LIN {X 0,Y 106.978,Z 615.98,A -85,B 0,C 180,E1 -26170.823,E2 -26170.823} C_VEL
LIN {X 0,Y 105.342,Z 616.584,A -85,B 0,C 180,E1 -26178.454,E2 -26178.454} C_VEL
LIN {X 0,Y 105.049,Z 615.86,A -85,B 0,C 180,E1 -26186.164,E2 -26186.164} C_VEL
LIN {X 0,Y 105.656,Z 613.825,A -85,B 0,C 180,E1 -26193.814,E2 -26193.814} C_VEL
LIN {X 0,Y 107.51,Z 610.427,A -85,B 0,C 180,E1 -26201.31,E2 -26201.31} C_VEL
LIN {X 0,Y 109.983,Z 606.946,A -85,B 0,C 180,E1 -26206.711,E2 -26206.711} C_VEL
LIN {X 0,Y 113.032,Z 602.521,A -85,B 0,C 180,E1 -26211.905,E2 -26211.905} C_VEL
LIN {X 0,Y 116.825,Z 597.145,A -85,B 0,C 180,E1 -26216.82,E2 -26216.82} C_VEL
LIN {X 0,Y 122.258,Z 589.447,A -85,B 0,C 180,E1 -26222.123,E2 -26222.123} C_VEL
LIN {X 0,Y 127.809,Z 581.397,A -85,B 0,C 180,E1 -26226.237,E2 -26226.237} C_VEL
LIN {X 0,Y 133.781,Z 571.709,A -85,B 0,C 180,E1 -26230.056,E2 -26230.056} C_VEL
LIN {X 0,Y 139.018,Z 562.033,A -85,B 0,C 180,E1 -26233.039,E2 -26233.039} C_VEL
LIN {X 0,Y 142.904,Z 554.154,A -85,B 0,C 180,E1 -26234.988,E2 -26234.988} C_VEL
LIN {X 0,Y 148.241,Z 542.028,A -85,B 0,C 180,E1 -26237.294,E2 -26237.294} C_VEL
LIN {X 0,Y 152.497,Z 530.39,A -85,B 0,C 180,E1 -26238.996,E2 -26238.996} C_VEL
LIN {X 0,Y 156.549,Z 516.515,A -85,B 0,C 180,E1 -26240.498,E2 -26240.498} C_VEL
LIN {X 0,Y 159.485,Z 502.683,A -85,B 0,C 180,E1 -26241.588,E2 -26241.588} C_VEL
LIN {X 0,Y 161.455,Z 488.768,A -85,B 0,C 180,E1 -26242.305,E2 -26242.305} C_VEL
LIN {X 0,Y 165.188,Z 446.212,A -85,B 0,C 180,E1 -26243.697,E2 -26243.697} C_VEL
LIN {X 0,Y 164.983,Z 444.977,A -85,B 0,C 180,E1 -26243.9,E2 -26243.9} C_VEL
LIN {X 0,Y 160.619,Z 435.797,A -85,B 0,C 180,E1 -26247.142,E2 -26247.142} C_VEL
LIN {X 0,Y 155.978,Z 427.263,A -85,B 0,C 180,E1 -26251.089,E2 -26251.089} C_VEL
LIN {X 0,Y 152.792,Z 421.962,A -85,B 0,C 180,E1 -26254.257,E2 -26254.257} C_VEL
LIN {X 0,Y 151.006,Z 419.154,A -85,B 0,C 180,E1 -26256.274,E2 -26256.274} C_VEL
LIN {X 0,Y 148.875,Z 415.814,A -85,B 0,C 180,E1 -26259.026,E2 -26259.026} C_VEL
LIN {X 0,Y 146.603,Z 412.142,A -85,B 0,C 180,E1 -26262.627,E2 -26262.627} C_VEL
LIN {X 0,Y 144.109,Z 408.852,A -85,B 0,C 180,E1 -26268.036,E2 -26268.036} C_VEL
LIN {X 0,Y 143.541,Z 407.096,A -85,B 0,C 180,E1 -26270.22,E2 -26270.22} C_VEL
LIN {X 0,Y 142.692,Z 406.337,A -85,B 0,C 180,E1 -26279.999,E2 -26279.999} C_VEL
LIN {X 0,Y 143.838,Z 407.423,A -85,B 0,C 180,E1 -26285.431,E2 -26285.431} C_VEL
LIN {X 0,Y 145.342,Z 410.732,A -85,B 0,C 180,E1 -26289.655,E2 -26289.655} C_VEL
LIN {X 0,Y 146.816,Z 412.43,A -85,B 0,C 180,E1 -26292.379,E2 -26292.379} C_VEL
LIN {X 0,Y 149.795,Z 417.149,A -85,B 0,C 180,E1 -26296.842,E2 -26296.842} C_VEL
LIN {X 0,Y 152.53,Z 421.521,A -85,B 0,C 180,E1 -26300.095,E2 -26300.095} C_VEL
LIN {X 0,Y 156.091,Z 427.345,A -85,B 0,C 180,E1 -26303.64,E2 -26303.64} C_VEL
LIN {X 0,Y 159.027,Z 432.919,A -85,B 0,C 180,E1 -26306.227,E2 -26306.227} C_VEL
LIN {X 0,Y 161.926,Z 440.414,A -85,B 0,C 180,E1 -26308.674,E2 -26308.674} C_VEL
LIN {X 0,Y 164.965,Z 449.328,A -85,B 0,C 180,E1 -26311.066,E2 -26311.066} C_VEL
LIN {X 0,Y 160.741,Z 497.527,A -85,B 0,C 180,E1 -26312.71,E2 -26312.71} C_VEL
LIN {X 0,Y 158.258,Z 511.944,A -85,B 0,C 180,E1 -26313.483,E2 -26313.483} C_VEL
LIN {X 0,Y 154.769,Z 525.923,A -85,B 0,C 180,E1 -26314.609,E2 -26314.609} C_VEL
LIN {X 0,Y 150.269,Z 539.82,A -85,B 0,C 180,E1 -26316.218,E2 -26316.218} C_VEL
LIN {X 0,Y 145.255,Z 552.264,A -85,B 0,C 180,E1 -26318.164,E2 -26318.164} C_VEL
LIN {X 0,Y 139.927,Z 563.656,A -85,B 0,C 180,E1 -26320.564,E2 -26320.564} C_VEL
LIN {X 0,Y 134.889,Z 573.146,A -85,B 0,C 180,E1 -26323.161,E2 -26323.161} C_VEL
LIN {X 0,Y 128.511,Z 583.722,A -85,B 0,C 180,E1 -26326.874,E2 -26326.874} C_VEL
LIN {X 0,Y 122.736,Z 592.445,A -85,B 0,C 180,E1 -26330.959,E2 -26330.959} C_VEL
LIN {X 0,Y 116.945,Z 600.809,A -85,B 0,C 180,E1 -26336.228,E2 -26336.228} C_VEL
LIN {X 0,Y 112.321,Z 607.529,A -85,B 0,C 180,E1 -26342.012,E2 -26342.012} C_VEL
LIN {X 0,Y 108.35,Z 613.483,A -85,B 0,C 180,E1 -26349.099,E2 -26349.099} C_VEL
LIN {X 0,Y 106.4,Z 616.926,A -85,B 0,C 180,E1 -26354.68,E2 -26354.68} C_VEL
LIN {X 0,Y 105.166,Z 620.167,A -85,B 0,C 180,E1 -26362.319,E2 -26362.319} C_VEL
LIN {X 0,Y 105.166,Z 622,A -85,B 0,C 180,E1 -26370,E2 -26370} C_VEL
LIN {X 0,Y 105.173,Z 622.449,A -85,B 0,C 180,E1 -26377.681,E2 -26377.681} C_VEL
LIN {X 0,Y 106.49,Z 621.572,A -85,B 0,C 180,E1 -26385.307,E2 -26385.307} C_VEL
LIN {X 0,Y 109.442,Z 619.368,A -85,B 0,C 180,E1 -26392.663,E2 -26392.663} C_VEL
LIN {X 0,Y 113.967,Z 615.782,A -85,B 0,C 180,E1 -26399.561,E2 -26399.561} C_VEL
LIN {X 0,Y 115.217,Z 614.69,A -85,B 0,C 180,E1 -26401.159,E2 -26401.159} C_VEL
LIN {X 0,Y 116.887,Z 612.823,A -85,B 0,C 180,E1 -26403.808,E2 -26403.808} C_VEL
LIN {X 0,Y 118.627,Z 609.391,A -85,B 0,C 180,E1 -26408.262,E2 -26408.262} C_VEL
LIN {X 0,Y 120.996,Z 605.387,A -85,B 0,C 180,E1 -26412.441,E2 -26412.441} C_VEL
LIN {X 0,Y 123.544,Z 602.626,A -85,B 0,C 180,E1 -26414.574,E2 -26414.574} C_VEL
LIN {X 0,Y 131.067,Z 595.341,A -85,B 0,C 180,E1 -26418.652,E2 -26418.652} C_VEL
LIN {X 0,Y 138.379,Z 587.385,A -85,B 0,C 180,E1 -26421.926,E2 -26421.926} C_VEL
LIN {X 0,Y 146.072,Z 577.81,A -85,B 0,C 180,E1 -26424.879,E2 -26424.879} C_VEL
LIN {X 0,Y 153.417,Z 567.213,A -85,B 0,C 180,E1 -26427.327,E2 -26427.327} C_VEL
LIN {X 0,Y 160.399,Z 555.509,A -85,B 0,C 180,E1 -26429.305,E2 -26429.305} C_VEL
LIN {X 0,Y 166.846,Z 542.503,A -85,B 0,C 180,E1 -26430.933,E2 -26430.933} C_VEL
LIN {X 0,Y 172,Z 529.708,A -85,B 0,C 180,E1 -26432.082,E2 -26432.082} C_VEL
LIN {X 0,Y 176.163,Z 516.241,A -85,B 0,C 180,E1 -26432.995,E2 -26432.995} C_VEL
LIN {X 0,Y 179.308,Z 502.034,A -85,B 0,C 180,E1 -26433.65,E2 -26433.65} C_VEL
LIN {X 0,Y 181.338,Z 486.524,A -85,B 0,C 180,E1 -26434.126,E2 -26434.126} C_VEL
LIN {X 0,Y 182.905,Z 469.902,A -85,B 0,C 180,E1 -26434.606,E2 -26434.606} C_VEL
LIN {X 0,Y 180.192,Z 461.706,A -85,B 0,C 180,E1 -26437.618,E2 -26437.618} C_VEL
LIN {X 0,Y 177.811,Z 455.265,A -85,B 0,C 180,E1 -26440.67,E2 -26440.67} C_VEL
LIN {X 0,Y 175.542,Z 451.014,A -85,B 0,C 180,E1 -26443.967,E2 -26443.967} C_VEL
LIN {X 0,Y 174.032,Z 448.052,A -85,B 0,C 180,E1 -26446.779,E2 -26446.779} C_VEL
LIN {X 0,Y 172.41,Z 444.514,A -85,B 0,C 180,E1 -26451.208,E2 -26451.208} C_VEL
LIN {X 0,Y 171.43,Z 443.369,A -85,B 0,C 180,E1 -26457.651,E2 -26457.651} C_VEL
LIN {X 0,Y 171.628,Z 443.532,A -85,B 0,C 180,E1 -26460.587,E2 -26460.587} C_VEL
LIN {X 0,Y 172.488,Z 444.731,A -85,B 0,C 180,E1 -26464.529,E2 -26464.529} C_VEL
LIN {X 0,Y 174.188,Z 448.243,A -85,B 0,C 180,E1 -26468.959,E2 -26468.959} C_VEL
LIN {X 0,Y 176.521,Z 452.894,A -85,B 0,C 180,E1 -26472.997,E2 -26472.997} C_VEL
LIN {X 0,Y 179.277,Z 458.182,A -85,B 0,C 180,E1 -26476.586,E2 -26476.586} C_VEL
LIN {X 0,Y 182.826,Z 465.868,A -85,B 0,C 180,E1 -26480.376,E2 -26480.376} C_VEL
LIN {X 0,Y 183.217,Z 466.787,A -85,B 0,C 180,E1 -26480.756,E2 -26480.756} C_VEL
LIN {X 0,Y 180.381,Z 493.857,A -85,B 0,C 180,E1 -26481.549,E2 -26481.549} C_VEL
LIN {X 0,Y 177.612,Z 508.239,A -85,B 0,C 180,E1 -26482.207,E2 -26482.207} C_VEL
LIN {X 0,Y 173.834,Z 521.809,A -85,B 0,C 180,E1 -26483.106,E2 -26483.106} C_VEL
LIN {X 0,Y 168.725,Z 535.471,A -85,B 0,C 180,E1 -26484.295,E2 -26484.295} C_VEL
LIN {X 0,Y 163.676,Z 546.452,A -85,B 0,C 180,E1 -26485.615,E2 -26485.615} C_VEL
LIN {X 0,Y 157.42,Z 557.978,A -85,B 0,C 180,E1 -26487.461,E2 -26487.461} C_VEL
LIN {X 0,Y 151.225,Z 567.55,A -85,B 0,C 180,E1 -26489.379,E2 -26489.379} C_VEL
LIN {X 0,Y 144.635,Z 576.544,A -85,B 0,C 180,E1 -26491.75,E2 -26491.75} C_VEL
LIN {X 0,Y 137.144,Z 585.567,A -85,B 0,C 180,E1 -26494.922,E2 -26494.922} C_VEL
LIN {X 0,Y 128.837,Z 594.174,A -85,B 0,C 180,E1 -26498.982,E2 -26498.982} C_VEL
LIN {X 0,Y 121.282,Z 601.093,A -85,B 0,C 180,E1 -26503.588,E2 -26503.588} C_VEL
LIN {X 0,Y 115.515,Z 605.855,A -85,B 0,C 180,E1 -26507.991,E2 -26507.991} C_VEL
LIN {X 0,Y 108.934,Z 610.764,A -85,B 0,C 180,E1 -26514.504,E2 -26514.504} C_VEL
LIN {X 0,Y 103.848,Z 614.157,A -85,B 0,C 180,E1 -26521.723,E2 -26521.723} C_VEL
LIN {X 0,Y 100.215,Z 616.148,A -85,B 0,C 180,E1 -26529.473,E2 -26529.473} C_VEL
LIN {X 0,Y 98.338,Z 616.788,A -85,B 0,C 180,E1 -26537.619,E2 -26537.619} C_VEL
LIN {X 0,Y 97.939,Z 616.099,A -85,B 0,C 180,E1 -26545.885,E2 -26545.885} C_VEL
LIN {X 0,Y 98.14,Z 615.26,A -85,B 0,C 180,E1 -26550,E2 -26550} C_VEL
LIN {X 0,Y 99.433,Z 612.582,A -85,B 0,C 180,E1 -26558.127,E2 -26558.127} C_VEL
LIN {X 0,Y 102.251,Z 608.494,A -85,B 0,C 180,E1 -26565.958,E2 -26565.958} C_VEL
LIN {X 0,Y 105.321,Z 604.462,A -85,B 0,C 180,E1 -26571.531,E2 -26571.531} C_VEL
LIN {X 0,Y 109.144,Z 599.427,A -85,B 0,C 180,E1 -26576.791,E2 -26576.791} C_VEL
LIN {X 0,Y 114.497,Z 592.249,A -85,B 0,C 180,E1 -26582.486,E2 -26582.486} C_VEL
LIN {X 0,Y 121.199,Z 583.338,A -85,B 0,C 180,E1 -26587.508,E2 -26587.508} C_VEL
LIN {X 0,Y 127.323,Z 574.006,A -85,B 0,C 180,E1 -26591.482,E2 -26591.482} C_VEL
LIN {X 0,Y 133.326,Z 563.687,A -85,B 0,C 180,E1 -26594.833,E2 -26594.833} C_VEL
LIN {X 0,Y 137.993,Z 554.781,A -85,B 0,C 180,E1 -26597.065,E2 -26597.065} C_VEL
LIN {X 0,Y 143.54,Z 542.777,A -85,B 0,C 180,E1 -26599.369,E2 -26599.369} C_VEL
LIN {X 0,Y 147.966,Z 531.241,A -85,B 0,C 180,E1 -26601.057,E2 -26601.057} C_VEL
LIN {X 0,Y 152.165,Z 517.653,A -85,B 0,C 180,E1 -26602.546,E2 -26602.546} C_VEL
LIN {X 0,Y 155.378,Z 503.296,A -85,B 0,C 180,E1 -26603.677,E2 -26603.677} C_VEL
LIN {X 0,Y 157.437,Z 489.422,A -85,B 0,C 180,E1 -26604.398,E2 -26604.398} C_VEL
LIN {X 0,Y 161.101,Z 449.238,A -85,B 0,C 180,E1 -26605.705,E2 -26605.705} C_VEL
LIN {X 0,Y 160.919,Z 447.991,A -85,B 0,C 180,E1 -26605.916,E2 -26605.916} C_VEL
LIN {X 0,Y 156.872,Z 439.376,A -85,B 0,C 180,E1 -26609.251,E2 -26609.251} C_VEL
LIN {X 0,Y 153.029,Z 432.072,A -85,B 0,C 180,E1 -26612.894,E2 -26612.894} C_VEL
LIN {X 0,Y 149.801,Z 426.345,A -85,B 0,C 180,E1 -26616.534,E2 -26616.534} C_VEL
LIN {X 0,Y 147.291,Z 422.35,A -85,B 0,C 180,E1 -26619.918,E2 -26619.918} C_VEL
LIN {X 0,Y 145.022,Z 418.618,A -85,B 0,C 180,E1 -26623.819,E2 -26623.819} C_VEL
LIN {X 0,Y 142.956,Z 415.552,A -85,B 0,C 180,E1 -26628.854,E2 -26628.854} C_VEL
LIN {X 0,Y 142.531,Z 414.075,A -85,B 0,C 180,E1 -26630.707,E2 -26630.707} C_VEL
LIN {X 0,Y 141.824,Z 413.393,A -85,B 0,C 180,E1 -26639.999,E2 -26639.999} C_VEL
LIN {X 0,Y 142.761,Z 414.272,A -85,B 0,C 180,E1 -26644.764,E2 -26644.764} C_VEL
LIN {X 0,Y 144.362,Z 417.845,A -85,B 0,C 180,E1 -26649.5,E2 -26649.5} C_VEL
LIN {X 0,Y 145.476,Z 419.202,A -85,B 0,C 180,E1 -26651.661,E2 -26651.661} C_VEL
LIN {X 0,Y 148.187,Z 423.711,A -85,B 0,C 180,E1 -26656.001,E2 -26656.001} C_VEL
LIN {X 0,Y 150.663,Z 427.94,A -85,B 0,C 180,E1 -26659.157,E2 -26659.157} C_VEL
LIN {X 0,Y 153.786,Z 433.303,A -85,B 0,C 180,E1 -26662.492,E2 -26662.492} C_VEL
LIN {X 0,Y 156.38,Z 438.493,A -85,B 0,C 180,E1 -26664.959,E2 -26664.959} C_VEL
LIN {X 0,Y 159.939,Z 448.587,A -85,B 0,C 180,E1 -26668.192,E2 -26668.192} C_VEL
LIN {X 0,Y 160.916,Z 451.729,A -85,B 0,C 180,E1 -26669.034,E2 -26669.034} C_VEL
LIN {X 0,Y 156.748,Z 497.427,A -85,B 0,C 180,E1 -26670.589,E2 -26670.589} C_VEL
LIN {X 0,Y 154.257,Z 511.481,A -85,B 0,C 180,E1 -26671.322,E2 -26671.322} C_VEL
LIN {X 0,Y 150.816,Z 524.958,A -85,B 0,C 180,E1 -26672.368,E2 -26672.368} C_VEL
LIN {X 0,Y 146.84,Z 537.25,A -85,B 0,C 180,E1 -26673.736,E2 -26673.736} C_VEL
LIN {X 0,Y 141.6,Z 550.147,A -85,B 0,C 180,E1 -26675.635,E2 -26675.635} C_VEL
LIN {X 0,Y 135.961,Z 561.87,A -85,B 0,C 180,E1 -26677.974,E2 -26677.974} C_VEL
LIN {X 0,Y 130.121,Z 572.617,A -85,B 0,C 180,E1 -26680.873,E2 -26680.873} C_VEL
LIN {X 0,Y 123.378,Z 583.245,A -85,B 0,C 180,E1 -26684.599,E2 -26684.599} C_VEL
LIN {X 0,Y 117.257,Z 592.014,A -85,B 0,C 180,E1 -26688.753,E2 -26688.753} C_VEL
LIN {X 0,Y 111.066,Z 600.428,A -85,B 0,C 180,E1 -26694.175,E2 -26694.175} C_VEL
LIN {X 0,Y 106.029,Z 607.187,A -85,B 0,C 180,E1 -26700.19,E2 -26700.19} C_VEL
LIN {X 0,Y 101.712,Z 613.176,A -85,B 0,C 180,E1 -26707.664,E2 -26707.664} C_VEL
LIN {X 0,Y 99.515,Z 616.637,A -85,B 0,C 180,E1 -26713.591,E2 -26713.591} C_VEL
LIN {X 0,Y 98.102,Z 619.917,A -85,B 0,C 180,E1 -26721.762,E2 -26721.762} C_VEL
LIN {X 0,Y 98.072,Z 621.779,A -85,B 0,C 180,E1 -26730,E2 -26730} C_VEL
LIN {X 0,Y 98.113,Z 622.254,A -85,B 0,C 180,E1 -26738.237,E2 -26738.237} C_VEL
LIN {X 0,Y 99.624,Z 621.403,A -85,B 0,C 180,E1 -26746.391,E2 -26746.391} C_VEL
LIN {X 0,Y 102.883,Z 619.226,A -85,B 0,C 180,E1 -26754.197,E2 -26754.197} C_VEL
LIN {X 0,Y 107.79,Z 615.668,A -85,B 0,C 180,E1 -26761.441,E2 -26761.441} C_VEL
LIN {X 0,Y 114.247,Z 610.629,A -85,B 0,C 180,E1 -26767.964,E2 -26767.964} C_VEL
LIN {X 0,Y 122.109,Z 603.966,A -85,B 0,C 180,E1 -26773.683,E2 -26773.683} C_VEL
LIN {X 0,Y 123.544,Z 602.626,A -85,B 0,C 180,E1 -26774.574,E2 -26774.574} C_VEL
LIN {X 0,Y 126.194,Z 599.722,A -85,B 0,C 180,E1 -26776.597,E2 -26776.597} C_VEL
LIN {X 0,Y 129.378,Z 594.686,A -85,B 0,C 180,E1 -26780.169,E2 -26780.169} C_VEL
LIN {X 0,Y 132.837,Z 589.224,A -85,B 0,C 180,E1 -26783.445,E2 -26783.445} C_VEL
LIN {X 0,Y 135.79,Z 585.532,A -85,B 0,C 180,E1 -26784.964,E2 -26784.964} C_VEL
LIN {X 0,Y 143.447,Z 576.129,A -85,B 0,C 180,E1 -26787.688,E2 -26787.688} C_VEL
LIN {X 0,Y 151.134,Z 565.237,A -85,B 0,C 180,E1 -26790.009,E2 -26790.009} C_VEL
LIN {X 0,Y 158.342,Z 553.168,A -85,B 0,C 180,E1 -26791.904,E2 -26791.904} C_VEL
LIN {X 0,Y 164.288,Z 541.252,A -85,B 0,C 180,E1 -26793.254,E2 -26793.254} C_VEL
LIN {X 0,Y 169.568,Z 528.127,A -85,B 0,C 180,E1 -26794.352,E2 -26794.352} C_VEL
LIN {X 0,Y 173.757,Z 514.407,A -85,B 0,C 180,E1 -26795.203,E2 -26795.203} C_VEL
LIN {X 0,Y 176.793,Z 500.293,A -85,B 0,C 180,E1 -26795.815,E2 -26795.815} C_VEL
LIN {X 0,Y 179.048,Z 482.171,A -85,B 0,C 180,E1 -26796.322,E2 -26796.322} C_VEL
LIN {X 0,Y 179.924,Z 473.211,A -85,B 0,C 180,E1 -26796.571,E2 -26796.571} C_VEL
LIN {X 0,Y 177.487,Z 465.387,A -85,B 0,C 180,E1 -26799.672,E2 -26799.672} C_VEL
LIN {X 0,Y 175.976,Z 461.216,A -85,B 0,C 180,E1 -26801.839,E2 -26801.839} C_VEL
LIN {X 0,Y 174.1,Z 457.474,A -85,B 0,C 180,E1 -26804.832,E2 -26804.832} C_VEL
LIN {X 0,Y 172.836,Z 454.794,A -85,B 0,C 180,E1 -26807.399,E2 -26807.399} C_VEL
LIN {X 0,Y 171.379,Z 451.415,A -85,B 0,C 180,E1 -26811.748,E2 -26811.748} C_VEL
LIN {X 0,Y 170.563,Z 450.423,A -85,B 0,C 180,E1 -26817.639,E2 -26817.639} C_VEL
LIN {X 0,Y 170.757,Z 450.614,A -85,B 0,C 180,E1 -26820.59,E2 -26820.59} C_VEL
LIN {X 0,Y 171.482,Z 451.693,A -85,B 0,C 180,E1 -26824.114,E2 -26824.114} C_VEL
LIN {X 0,Y 173.28,Z 455.722,A -85,B 0,C 180,E1 -26829.006,E2 -26829.006} C_VEL
LIN {X 0,Y 175.2,Z 459.749,A -85,B 0,C 180,E1 -26832.452,E2 -26832.452} C_VEL
LIN {X 0,Y 177.515,Z 464.469,A -85,B 0,C 180,E1 -26835.676,E2 -26835.676} C_VEL
LIN {X 0,Y 180.167,Z 470.555,A -85,B 0,C 180,E1 -26838.778,E2 -26838.778} C_VEL
LIN {X 0,Y 177.56,Z 494.301,A -85,B 0,C 180,E1 -26839.467,E2 -26839.467} C_VEL
LIN {X 0,Y 174.687,Z 508.753,A -85,B 0,C 180,E1 -26840.114,E2 -26840.114} C_VEL
LIN {X 0,Y 170.779,Z 522.33,A -85,B 0,C 180,E1 -26840.987,E2 -26840.987} C_VEL
LIN {X 0,Y 165.81,Z 535.301,A -85,B 0,C 180,E1 -26842.079,E2 -26842.079} C_VEL
LIN {X 0,Y 159.976,Z 547.572,A -85,B 0,C 180,E1 -26843.497,E2 -26843.497} C_VEL
LIN {X 0,Y 153.533,Z 558.935,A -85,B 0,C 180,E1 -26845.302,E2 -26845.302} C_VEL
LIN {X 0,Y 146.433,Z 569.358,A -85,B 0,C 180,E1 -26847.388,E2 -26847.388} C_VEL
LIN {X 0,Y 138.319,Z 579.704,A -85,B 0,C 180,E1 -26850.256,E2 -26850.256} C_VEL
LIN {X 0,Y 130.633,Z 588.224,A -85,B 0,C 180,E1 -26853.498,E2 -26853.498} C_VEL
LIN {X 0,Y 122.068,Z 596.332,A -85,B 0,C 180,E1 -26857.659,E2 -26857.659} C_VEL
LIN {X 0,Y 113.892,Z 603.166,A -85,B 0,C 180,E1 -26862.75,E2 -26862.75} C_VEL
LIN {X 0,Y 106.518,Z 608.597,A -85,B 0,C 180,E1 -26868.715,E2 -26868.715} C_VEL
LIN {X 0,Y 100.144,Z 612.764,A -85,B 0,C 180,E1 -26875.845,E2 -26875.845} C_VEL
LIN {X 0,Y 95.319,Z 615.476,A -85,B 0,C 180,E1 -26883.743,E2 -26883.743} C_VEL
LIN {X 0,Y 92.168,Z 616.819,A -85,B 0,C 180,E1 -26892.241,E2 -26892.241} C_VEL
LIN {X 0,Y 90.928,Z 616.826,A -85,B 0,C 180,E1 -26901.107,E2 -26901.107} C_VEL
LIN {X 0,Y 90.828,Z 616.334,A -85,B 0,C 180,E1 -26905.562,E2 -26905.562} C_VEL
LIN {X 0,Y 91.044,Z 615.512,A -85,B 0,C 180,E1 -26910,E2 -26910} C_VEL
LIN {X 0,Y 92.441,Z 612.864,A -85,B 0,C 180,E1 -26918.746,E2 -26918.746} C_VEL
LIN {X 0,Y 95.457,Z 608.807,A -85,B 0,C 180,E1 -26927.128,E2 -26927.128} C_VEL
LIN {X 0,Y 98.764,Z 604.799,A -85,B 0,C 180,E1 -26933.04,E2 -26933.04} C_VEL
LIN {X 0,Y 102.861,Z 599.792,A -85,B 0,C 180,E1 -26938.573,E2 -26938.573} C_VEL
LIN {X 0,Y 108.598,Z 592.652,A -85,B 0,C 180,E1 -26944.49,E2 -26944.49} C_VEL
LIN {X 0,Y 115.681,Z 583.797,A -85,B 0,C 180,E1 -26949.636,E2 -26949.636} C_VEL
LIN {X 0,Y 122.122,Z 574.527,A -85,B 0,C 180,E1 -26953.677,E2 -26953.677} C_VEL
LIN {X 0,Y 128.41,Z 564.276,A -85,B 0,C 180,E1 -26957.057,E2 -26957.057} C_VEL
LIN {X 0,Y 133.278,Z 555.407,A -85,B 0,C 180,E1 -26959.29,E2 -26959.29} C_VEL
LIN {X 0,Y 139.05,Z 543.498,A -85,B 0,C 180,E1 -26961.575,E2 -26961.575} C_VEL
LIN {X 0,Y 143.635,Z 532.081,A -85,B 0,C 180,E1 -26963.247,E2 -26963.247} C_VEL
LIN {X 0,Y 147.98,Z 518.717,A -85,B 0,C 180,E1 -26964.715,E2 -26964.715} C_VEL
LIN {X 0,Y 151.315,Z 504.817,A -85,B 0,C 180,E1 -26965.825,E2 -26965.825} C_VEL
LIN {X 0,Y 153.645,Z 490.117,A -85,B 0,C 180,E1 -26966.59,E2 -26966.59} C_VEL
LIN {X 0,Y 157.258,Z 451.619,A -85,B 0,C 180,E1 -26967.851,E2 -26967.851} C_VEL
LIN {X 0,Y 153.572,Z 443.488,A -85,B 0,C 180,E1 -26971.231,E2 -26971.231} C_VEL
LIN {X 0,Y 149.74,Z 435.854,A -85,B 0,C 180,E1 -26975.362,E2 -26975.362} C_VEL
LIN {X 0,Y 147.457,Z 431.908,A -85,B 0,C 180,E1 -26978.258,E2 -26978.258} C_VEL
LIN {X 0,Y 145.816,Z 428.996,A -85,B 0,C 180,E1 -26980.714,E2 -26980.714} C_VEL
LIN {X 0,Y 143.639,Z 425.279,A -85,B 0,C 180,E1 -26984.752,E2 -26984.752} C_VEL
LIN {X 0,Y 141.841,Z 422.276,A -85,B 0,C 180,E1 -26989.652,E2 -26989.652} C_VEL
LIN {X 0,Y 141.478,Z 421.011,A -85,B 0,C 180,E1 -26991.429,E2 -26991.429} C_VEL
LIN {X 0,Y 140.955,Z 420.453,A -85,B 0,C 180,E1 -26999.999,E2 -26999.999} C_VEL
LIN {X 0,Y 141.765,Z 421.374,A -85,B 0,C 180,E1 -27004.397,E2 -27004.397} C_VEL
LIN {X 0,Y 143.385,Z 424.945,A -85,B 0,C 180,E1 -27009.343,E2 -27009.343} C_VEL
LIN {X 0,Y 144.137,Z 425.963,A -85,B 0,C 180,E1 -27010.89,E2 -27010.89} C_VEL
LIN {X 0,Y 146.71,Z 430.515,A -85,B 0,C 180,E1 -27015.298,E2 -27015.298} C_VEL
LIN {X 0,Y 148.93,Z 434.483,A -85,B 0,C 180,E1 -27018.306,E2 -27018.306} C_VEL
LIN {X 0,Y 152.01,Z 440.251,A -85,B 0,C 180,E1 -27021.813,E2 -27021.813} C_VEL
LIN {X 0,Y 153.809,Z 444.149,A -85,B 0,C 180,E1 -27023.655,E2 -27023.655} C_VEL
LIN {X 0,Y 156.887,Z 453.647,A -85,B 0,C 180,E1 -27026.731,E2 -27026.731} C_VEL
LIN {X 0,Y 157.108,Z 454.381,A -85,B 0,C 180,E1 -27026.942,E2 -27026.942} C_VEL
LIN {X 0,Y 152.938,Z 497.627,A -85,B 0,C 180,E1 -27028.374,E2 -27028.374} C_VEL
LIN {X 0,Y 150.319,Z 511.787,A -85,B 0,C 180,E1 -27029.106,E2 -27029.106} C_VEL
LIN {X 0,Y 146.772,Z 525.133,A -85,B 0,C 180,E1 -27030.128,E2 -27030.128} C_VEL
LIN {X 0,Y 142.317,Z 538.232,A -85,B 0,C 180,E1 -27031.586,E2 -27031.586} C_VEL
LIN {X 0,Y 136.898,Z 550.901,A -85,B 0,C 180,E1 -27033.463,E2 -27033.463} C_VEL
LIN {X 0,Y 131.045,Z 562.456,A -85,B 0,C 180,E1 -27035.79,E2 -27035.79} C_VEL
LIN {X 0,Y 125.57,Z 572.087,A -85,B 0,C 180,E1 -27038.412,E2 -27038.412} C_VEL
LIN {X 0,Y 118.471,Z 582.768,A -85,B 0,C 180,E1 -27042.138,E2 -27042.138} C_VEL
LIN {X 0,Y 111.956,Z 591.581,A -85,B 0,C 180,E1 -27046.328,E2 -27046.328} C_VEL
LIN {X 0,Y 105.36,Z 600.043,A -85,B 0,C 180,E1 -27051.901,E2 -27051.901} C_VEL
LIN {X 0,Y 99.753,Z 606.984,A -85,B 0,C 180,E1 -27058.3,E2 -27058.3} C_VEL
LIN {X 0,Y 95.149,Z 612.87,A -85,B 0,C 180,E1 -27066.031,E2 -27066.031} C_VEL
LIN {X 0,Y 92.678,Z 616.345,A -85,B 0,C 180,E1 -27072.342,E2 -27072.342} C_VEL
LIN {X 0,Y 91.065,Z 619.665,A -85,B 0,C 180,E1 -27081.121,E2 -27081.121} C_VEL
LIN {X 0,Y 90.97,Z 621.557,A -85,B 0,C 180,E1 -27090,E2 -27090} C_VEL
LIN {X 0,Y 90.862,Z 621.975,A -85,B 0,C 180,E1 -27094.436,E2 -27094.436} C_VEL
LIN {X 0,Y 91.733,Z 621.811,A -85,B 0,C 180,E1 -27103.288,E2 -27103.288} C_VEL
LIN {X 0,Y 94.31,Z 620.325,A -85,B 0,C 180,E1 -27111.876,E2 -27111.876} C_VEL
LIN {X 0,Y 98.874,Z 617.497,A -85,B 0,C 180,E1 -27119.839,E2 -27119.839} C_VEL
LIN {X 0,Y 105.007,Z 613.242,A -85,B 0,C 180,E1 -27127.04,E2 -27127.04} C_VEL
LIN {X 0,Y 112.725,Z 607.445,A -85,B 0,C 180,E1 -27133.3,E2 -27133.3} C_VEL
LIN {X 0,Y 120.445,Z 600.935,A -85,B 0,C 180,E1 -27138.071,E2 -27138.071} C_VEL
LIN {X 0,Y 128.999,Z 592.88,A -85,B 0,C 180,E1 -27142.184,E2 -27142.184} C_VEL
LIN {X 0,Y 135.79,Z 585.532,A -85,B 0,C 180,E1 -27144.964,E2 -27144.964} C_VEL
LIN {X 0,Y 138.742,Z 581.719,A -85,B 0,C 180,E1 -27146.385,E2 -27146.385} C_VEL
LIN {X 0,Y 142.383,Z 575.326,A -85,B 0,C 180,E1 -27149.094,E2 -27149.094} C_VEL
LIN {X 0,Y 145.943,Z 568.505,A -85,B 0,C 180,E1 -27151.576,E2 -27151.576} C_VEL
LIN {X 0,Y 148.656,Z 564.023,A -85,B 0,C 180,E1 -27152.632,E2 -27152.632} C_VEL
LIN {X 0,Y 155.893,Z 552.062,A -85,B 0,C 180,E1 -27154.376,E2 -27154.376} C_VEL
LIN {X 0,Y 161.997,Z 539.914,A -85,B 0,C 180,E1 -27155.653,E2 -27155.653} C_VEL
LIN {X 0,Y 167.386,Z 526.439,A -85,B 0,C 180,E1 -27156.703,E2 -27156.703} C_VEL
LIN {X 0,Y 171.682,Z 512.225,A -85,B 0,C 180,E1 -27157.494,E2 -27157.494} C_VEL
LIN {X 0,Y 174.68,Z 497.787,A -85,B 0,C 180,E1 -27158.051,E2 -27158.051} C_VEL
LIN {X 0,Y 177.125,Z 476.542,A -85,B 0,C 180,E1 -27158.633,E2 -27158.633} C_VEL
LIN {X 0,Y 175.113,Z 469.694,A -85,B 0,C 180,E1 -27161.588,E2 -27161.588} C_VEL
LIN {X 0,Y 174.327,Z 467.447,A -85,B 0,C 180,E1 -27162.855,E2 -27162.855} C_VEL
LIN {X 0,Y 172.77,Z 464.08,A -85,B 0,C 180,E1 -27165.573,E2 -27165.573} C_VEL
LIN {X 0,Y 171.589,Z 461.48,A -85,B 0,C 180,E1 -27168.183,E2 -27168.183} C_VEL
LIN {X 0,Y 170.379,Z 458.353,A -85,B 0,C 180,E1 -27172.223,E2 -27172.223} C_VEL
LIN {X 0,Y 169.696,Z 457.476,A -85,B 0,C 180,E1 -27177.627,E2 -27177.627} C_VEL
LIN {X 0,Y 169.89,Z 457.663,A -85,B 0,C 180,E1 -27180.593,E2 -27180.593} C_VEL
LIN {X 0,Y 170.487,Z 458.64,A -85,B 0,C 180,E1 -27183.694,E2 -27183.694} C_VEL
LIN {X 0,Y 172.152,Z 462.655,A -85,B 0,C 180,E1 -27188.567,E2 -27188.567} C_VEL
LIN {X 0,Y 174.064,Z 466.899,A -85,B 0,C 180,E1 -27192.165,E2 -27192.165} C_VEL
LIN {X 0,Y 176.541,Z 472.515,A -85,B 0,C 180,E1 -27195.741,E2 -27195.741} C_VEL
LIN {X 0,Y 177.309,Z 474.419,A -85,B 0,C 180,E1 -27196.718,E2 -27196.718} C_VEL
LIN {X 0,Y 174.87,Z 495.427,A -85,B 0,C 180,E1 -27197.347,E2 -27197.347} C_VEL
LIN {X 0,Y 171.851,Z 509.857,A -85,B 0,C 180,E1 -27197.981,E2 -27197.981} C_VEL
LIN {X 0,Y 167.573,Z 523.987,A -85,B 0,C 180,E1 -27198.866,E2 -27198.866} C_VEL
LIN {X 0,Y 162.406,Z 536.817,A -85,B 0,C 180,E1 -27199.925,E2 -27199.925} C_VEL
LIN {X 0,Y 156.392,Z 548.916,A -85,B 0,C 180,E1 -27201.317,E2 -27201.317} C_VEL
LIN {X 0,Y 149.14,Z 560.985,A -85,B 0,C 180,E1 -27203.232,E2 -27203.232} C_VEL
LIN {X 0,Y 141.839,Z 571.099,A -85,B 0,C 180,E1 -27205.273,E2 -27205.273} C_VEL
LIN {X 0,Y 133.91,Z 580.646,A -85,B 0,C 180,E1 -27207.946,E2 -27207.946} C_VEL
LIN {X 0,Y 125.488,Z 589.442,A -85,B 0,C 180,E1 -27211.341,E2 -27211.341} C_VEL
LIN {X 0,Y 116.588,Z 597.361,A -85,B 0,C 180,E1 -27215.532,E2 -27215.532} C_VEL
LIN {X 0,Y 108.531,Z 603.651,A -85,B 0,C 180,E1 -27220.359,E2 -27220.359} C_VEL
LIN {X 0,Y 101.225,Z 608.687,A -85,B 0,C 180,E1 -27226.028,E2 -27226.028} C_VEL
LIN {X 0,Y 94.267,Z 612.887,A -85,B 0,C 180,E1 -27233.385,E2 -27233.385} C_VEL
LIN {X 0,Y 88.938,Z 615.628,A -85,B 0,C 180,E1 -27241.697,E2 -27241.697} C_VEL
LIN {X 0,Y 85.357,Z 617.001,A -85,B 0,C 180,E1 -27250.77,E2 -27250.77} C_VEL
LIN {X 0,Y 83.866,Z 617.039,A -85,B 0,C 180,E1 -27260.351,E2 -27260.351} C_VEL
LIN {X 0,Y 83.741,Z 616.564,A -85,B 0,C 180,E1 -27265.186,E2 -27265.186} C_VEL
LIN {X 0,Y 83.94,Z 615.761,A -85,B 0,C 180,E1 -27270,E2 -27270} C_VEL
LIN {X 0,Y 85.445,Z 613.146,A -85,B 0,C 180,E1 -27279.468,E2 -27279.468} C_VEL
LIN {X 0,Y 88.715,Z 609.121,A -85,B 0,C 180,E1 -27288.474,E2 -27288.474} C_VEL
LIN {X 0,Y 93.672,Z 603.562,A -85,B 0,C 180,E1 -27296.754,E2 -27296.754} C_VEL
LIN {X 0,Y 98.335,Z 598.296,A -85,B 0,C 180,E1 -27302.413,E2 -27302.413} C_VEL
LIN {X 0,Y 104.892,Z 590.718,A -85,B 0,C 180,E1 -27308.3,E2 -27308.3} C_VEL
LIN {X 0,Y 111.419,Z 582.805,A -85,B 0,C 180,E1 -27312.694,E2 -27312.694} C_VEL
LIN {X 0,Y 118.335,Z 573.278,A -85,B 0,C 180,E1 -27316.681,E2 -27316.681} C_VEL
LIN {X 0,Y 124.367,Z 563.795,A -85,B 0,C 180,E1 -27319.72,E2 -27319.72} C_VEL
LIN {X 0,Y 128.099,Z 557.201,A -85,B 0,C 180,E1 -27321.427,E2 -27321.427} C_VEL
LIN {X 0,Y 134.102,Z 545.627,A -85,B 0,C 180,E1 -27323.685,E2 -27323.685} C_VEL
LIN {X 0,Y 139.519,Z 532.916,A -85,B 0,C 180,E1 -27325.575,E2 -27325.575} C_VEL
LIN {X 0,Y 144.028,Z 519.724,A -85,B 0,C 180,E1 -27327.002,E2 -27327.002} C_VEL
LIN {X 0,Y 147.641,Z 505.395,A -85,B 0,C 180,E1 -27328.146,E2 -27328.146} C_VEL
LIN {X 0,Y 149.962,Z 491.732,A -85,B 0,C 180,E1 -27328.867,E2 -27328.867} C_VEL
LIN {X 0,Y 153.585,Z 454.813,A -85,B 0,C 180,E1 -27330.061,E2 -27330.061} C_VEL
LIN {X 0,Y 150.418,Z 447.565,A -85,B 0,C 180,E1 -27333.337,E2 -27333.337} C_VEL
LIN {X 0,Y 147.242,Z 441.062,A -85,B 0,C 180,E1 -27337.186,E2 -27337.186} C_VEL
LIN {X 0,Y 144.574,Z 435.911,A -85,B 0,C 180,E1 -27341.194,E2 -27341.194} C_VEL
LIN {X 0,Y 142.452,Z 432.127,A -85,B 0,C 180,E1 -27345.353,E2 -27345.353} C_VEL
LIN {X 0,Y 140.751,Z 428.988,A -85,B 0,C 180,E1 -27350.479,E2 -27350.479} C_VEL
LIN {X 0,Y 140.528,Z 428.012,A -85,B 0,C 180,E1 -27351.775,E2 -27351.775} C_VEL
LIN {X 0,Y 140.087,Z 427.514,A -85,B 0,C 180,E1 -27359.999,E2 -27359.999} C_VEL
LIN {X 0,Y 140.726,Z 428.262,A -85,B 0,C 180,E1 -27363.757,E2 -27363.757} C_VEL
LIN {X 0,Y 142.162,Z 431.687,A -85,B 0,C 180,E1 -27368.608,E2 -27368.608} C_VEL
LIN {X 0,Y 142.898,Z 432.833,A -85,B 0,C 180,E1 -27370.26,E2 -27370.26} C_VEL
LIN {X 0,Y 145.103,Z 437.004,A -85,B 0,C 180,E1 -27374.336,E2 -27374.336} C_VEL
LIN {X 0,Y 147.192,Z 440.994,A -85,B 0,C 180,E1 -27377.39,E2 -27377.39} C_VEL
LIN {X 0,Y 150.154,Z 446.933,A -85,B 0,C 180,E1 -27380.998,E2 -27380.998} C_VEL
LIN {X 0,Y 151.552,Z 450.518,A -85,B 0,C 180,E1 -27382.574,E2 -27382.574} C_VEL
LIN {X 0,Y 153.45,Z 456.893,A -85,B 0,C 180,E1 -27384.687,E2 -27384.687} C_VEL
LIN {X 0,Y 149.496,Z 497.047,A -85,B 0,C 180,E1 -27386.023,E2 -27386.023} C_VEL
LIN {X 0,Y 146.805,Z 511.318,A -85,B 0,C 180,E1 -27386.73,E2 -27386.73} C_VEL
LIN {X 0,Y 142.959,Z 525.299,A -85,B 0,C 180,E1 -27387.76,E2 -27387.76} C_VEL
LIN {X 0,Y 138.711,Z 537.43,A -85,B 0,C 180,E1 -27389.073,E2 -27389.073} C_VEL
LIN {X 0,Y 133.102,Z 550.217,A -85,B 0,C 180,E1 -27390.904,E2 -27390.904} C_VEL
LIN {X 0,Y 126.993,Z 561.855,A -85,B 0,C 180,E1 -27393.171,E2 -27393.171} C_VEL
LIN {X 0,Y 119.983,Z 573.522,A -85,B 0,C 180,E1 -27396.35,E2 -27396.35} C_VEL
LIN {X 0,Y 112.606,Z 583.923,A -85,B 0,C 180,E1 -27400.133,E2 -27400.133} C_VEL
LIN {X 0,Y 105.832,Z 592.51,A -85,B 0,C 180,E1 -27404.448,E2 -27404.448} C_VEL
LIN {X 0,Y 98.878,Z 600.713,A -85,B 0,C 180,E1 -27410.231,E2 -27410.231} C_VEL
LIN {X 0,Y 94.063,Z 606.211,A -85,B 0,C 180,E1 -27415.521,E2 -27415.521} C_VEL
LIN {X 0,Y 89.789,Z 611.19,A -85,B 0,C 180,E1 -27421.99,E2 -27421.99} C_VEL
LIN {X 0,Y 85.874,Z 616.052,A -85,B 0,C 180,E1 -27430.891,E2 -27430.891} C_VEL
LIN {X 0,Y 84.026,Z 619.409,A -85,B 0,C 180,E1 -27440.37,E2 -27440.37} C_VEL
LIN {X 0,Y 83.876,Z 621.336,A -85,B 0,C 180,E1 -27450,E2 -27450} C_VEL
LIN {X 0,Y 83.776,Z 621.767,A -85,B 0,C 180,E1 -27454.812,E2 -27454.812} C_VEL
LIN {X 0,Y 84.797,Z 621.629,A -85,B 0,C 180,E1 -27464.397,E2 -27464.397} C_VEL
LIN {X 0,Y 87.725,Z 620.17,A -85,B 0,C 180,E1 -27473.614,E2 -27473.614} C_VEL
LIN {X 0,Y 92.737,Z 617.369,A -85,B 0,C 180,E1 -27482.039,E2 -27482.039} C_VEL
LIN {X 0,Y 99.402,Z 613.144,A -85,B 0,C 180,E1 -27489.519,E2 -27489.519} C_VEL
LIN {X 0,Y 107.65,Z 607.378,A -85,B 0,C 180,E1 -27495.902,E2 -27495.902} C_VEL
LIN {X 0,Y 115.806,Z 600.904,A -85,B 0,C 180,E1 -27500.694,E2 -27500.694} C_VEL
LIN {X 0,Y 124.771,Z 592.886,A -85,B 0,C 180,E1 -27504.761,E2 -27504.761} C_VEL
LIN {X 0,Y 133.876,Z 583.371,A -85,B 0,C 180,E1 -27508.192,E2 -27508.192} C_VEL
LIN {X 0,Y 142.616,Z 572.533,A -85,B 0,C 180,E1 -27511.011,E2 -27511.011} C_VEL
LIN {X 0,Y 148.656,Z 564.023,A -85,B 0,C 180,E1 -27512.632,E2 -27512.632} C_VEL
LIN {X 0,Y 151.327,Z 559.403,A -85,B 0,C 180,E1 -27513.609,E2 -27513.609} C_VEL
LIN {X 0,Y 154.696,Z 551.76,A -85,B 0,C 180,E1 -27515.616,E2 -27515.616} C_VEL
LIN {X 0,Y 157.795,Z 543.776,A -85,B 0,C 180,E1 -27517.434,E2 -27517.434} C_VEL
LIN {X 0,Y 159.95,Z 538.627,A -85,B 0,C 180,E1 -27518.12,E2 -27518.12} C_VEL
LIN {X 0,Y 165.485,Z 524.754,A -85,B 0,C 180,E1 -27519.12,E2 -27519.12} C_VEL
LIN {X 0,Y 169.733,Z 510.611,A -85,B 0,C 180,E1 -27519.822,E2 -27519.822} C_VEL
LIN {X 0,Y 172.659,Z 496.278,A -85,B 0,C 180,E1 -27520.317,E2 -27520.317} C_VEL
LIN {X 0,Y 174.544,Z 479.975,A -85,B 0,C 180,E1 -27520.764,E2 -27520.764} C_VEL
LIN {X 0,Y 172.981,Z 474.182,A -85,B 0,C 180,E1 -27523.478,E2 -27523.478} C_VEL
LIN {X 0,Y 171.381,Z 470.486,A -85,B 0,C 180,E1 -27526.513,E2 -27526.513} C_VEL
LIN {X 0,Y 170.424,Z 468.219,A -85,B 0,C 180,E1 -27528.855,E2 -27528.855} C_VEL
LIN {X 0,Y 169.357,Z 465.263,A -85,B 0,C 180,E1 -27532.849,E2 -27532.849} C_VEL
LIN {X 0,Y 168.831,Z 464.521,A -85,B 0,C 180,E1 -27537.615,E2 -27537.615} C_VEL
LIN {X 0,Y 169.072,Z 464.866,A -85,B 0,C 180,E1 -27541.02,E2 -27541.02} C_VEL
LIN {X 0,Y 169.499,Z 465.61,A -85,B 0,C 180,E1 -27543.269,E2 -27543.269} C_VEL
LIN {X 0,Y 170.911,Z 469.308,A -85,B 0,C 180,E1 -27547.829,E2 -27547.829} C_VEL
LIN {X 0,Y 172.607,Z 473.398,A -85,B 0,C 180,E1 -27551.329,E2 -27551.329} C_VEL
LIN {X 0,Y 174.695,Z 478.434,A -85,B 0,C 180,E1 -27554.622,E2 -27554.622} C_VEL
LIN {X 0,Y 172.346,Z 497.089,A -85,B 0,C 180,E1 -27555.193,E2 -27555.193} C_VEL
LIN {X 0,Y 169.223,Z 511.13,A -85,B 0,C 180,E1 -27555.792,E2 -27555.792} C_VEL
LIN {X 0,Y 165.005,Z 524.507,A -85,B 0,C 180,E1 -27556.596,E2 -27556.596} C_VEL
LIN {X 0,Y 159.249,Z 538.251,A -85,B 0,C 180,E1 -27557.691,E2 -27557.691} C_VEL
LIN {X 0,Y 153.25,Z 549.825,A -85,B 0,C 180,E1 -27558.99,E2 -27558.99} C_VEL
LIN {X 0,Y 145.706,Z 561.875,A -85,B 0,C 180,E1 -27560.845,E2 -27560.845} C_VEL
LIN {X 0,Y 137.448,Z 572.768,A -85,B 0,C 180,E1 -27563.017,E2 -27563.017} C_VEL
LIN {X 0,Y 129.422,Z 581.914,A -85,B 0,C 180,E1 -27565.596,E2 -27565.596} C_VEL
LIN {X 0,Y 120.535,Z 590.656,A -85,B 0,C 180,E1 -27569.001,E2 -27569.001} C_VEL
LIN {X 0,Y 111.284,Z 598.39,A -85,B 0,C 180,E1 -27573.197,E2 -27573.197} C_VEL
LIN {X 0,Y 103.382,Z 604.134,A -85,B 0,C 180,E1 -27577.723,E2 -27577.723} C_VEL
LIN {X 0,Y 96.173,Z 608.778,A -85,B 0,C 180,E1 -27583.049,E2 -27583.049} C_VEL
LIN {X 0,Y 88.586,Z 613.01,A -85,B 0,C 180,E1 -27590.603,E2 -27590.603} C_VEL
LIN {X 0,Y 82.69,Z 615.781,A -85,B 0,C 180,E1 -27599.339,E2 -27599.339} C_VEL
LIN {X 0,Y 78.612,Z 617.183,A -85,B 0,C 180,E1 -27609.047,E2 -27609.047} C_VEL
LIN {X 0,Y 76.833,Z 617.249,A -85,B 0,C 180,E1 -27619.459,E2 -27619.459} C_VEL
LIN {X 0,Y 76.63,Z 616.791,A -85,B 0,C 180,E1 -27624.738,E2 -27624.738} C_VEL
LIN {X 0,Y 76.844,Z 616.004,A -85,B 0,C 180,E1 -27630,E2 -27630} C_VEL
LIN {X 0,Y 78.466,Z 613.427,A -85,B 0,C 180,E1 -27640.319,E2 -27640.319} C_VEL
LIN {X 0,Y 82.031,Z 609.433,A -85,B 0,C 180,E1 -27650.041,E2 -27650.041} C_VEL
LIN {X 0,Y 85.916,Z 605.46,A -85,B 0,C 180,E1 -27656.738,E2 -27656.738} C_VEL
LIN {X 0,Y 90.664,Z 600.522,A -85,B 0,C 180,E1 -27662.862,E2 -27662.862} C_VEL
LIN {X 0,Y 97.277,Z 593.455,A -85,B 0,C 180,E1 -27669.21,E2 -27669.21} C_VEL
LIN {X 0,Y 105.163,Z 584.692,A -85,B 0,C 180,E1 -27674.564,E2 -27674.564} C_VEL
LIN {X 0,Y 112.335,Z 575.532,A -85,B 0,C 180,E1 -27678.656,E2 -27678.656} C_VEL
LIN {X 0,Y 119.234,Z 565.425,A -85,B 0,C 180,E1 -27682.033,E2 -27682.033} C_VEL
LIN {X 0,Y 123.817,Z 557.822,A -85,B 0,C 180,E1 -27683.984,E2 -27683.984} C_VEL
LIN {X 0,Y 130.05,Z 546.337,A -85,B 0,C 180,E1 -27686.19,E2 -27686.19} C_VEL
LIN {X 0,Y 135.652,Z 533.748,A -85,B 0,C 180,E1 -27688.035,E2 -27688.035} C_VEL
LIN {X 0,Y 140.313,Z 520.732,A -85,B 0,C 180,E1 -27689.417,E2 -27689.417} C_VEL
LIN {X 0,Y 144.052,Z 506.707,A -85,B 0,C 180,E1 -27690.524,E2 -27690.524} C_VEL
LIN {X 0,Y 146.682,Z 492.166,A -85,B 0,C 180,E1 -27691.284,E2 -27691.284} C_VEL
LIN {X 0,Y 150.148,Z 458.115,A -85,B 0,C 180,E1 -27692.367,E2 -27692.367} C_VEL
LIN {X 0,Y 146.886,Z 450.447,A -85,B 0,C 180,E1 -27696.276,E2 -27696.276} C_VEL
LIN {X 0,Y 144.495,Z 445.364,A -85,B 0,C 180,E1 -27699.706,E2 -27699.706} C_VEL
LIN {X 0,Y 142.705,Z 441.868,A -85,B 0,C 180,E1 -27702.812,E2 -27702.812} C_VEL
LIN {X 0,Y 141.168,Z 438.847,A -85,B 0,C 180,E1 -27706.229,E2 -27706.229} C_VEL
LIN {X 0,Y 139.63,Z 435.385,A -85,B 0,C 180,E1 -27711.722,E2 -27711.722} C_VEL
LIN {X 0,Y 139.578,Z 435.062,A -85,B 0,C 180,E1 -27712.126,E2 -27712.126} C_VEL
LIN {X 0,Y 139.219,Z 434.573,A -85,B 0,C 180,E1 -27719.999,E2 -27719.999} C_VEL
LIN {X 0,Y 139.73,Z 435.223,A -85,B 0,C 180,E1 -27723.243,E2 -27723.243} C_VEL
LIN {X 0,Y 141.176,Z 438.776,A -85,B 0,C 180,E1 -27728.408,E2 -27728.408} C_VEL
LIN {X 0,Y 143.218,Z 442.713,A -85,B 0,C 180,E1 -27732.757,E2 -27732.757} C_VEL
LIN {X 0,Y 145.401,Z 447.296,A -85,B 0,C 180,E1 -27736.316,E2 -27736.316} C_VEL
LIN {X 0,Y 148.075,Z 453.032,A -85,B 0,C 180,E1 -27739.855,E2 -27739.855} C_VEL
LIN {X 0,Y 149.543,Z 457.722,A -85,B 0,C 180,E1 -27741.721,E2 -27741.721} C_VEL
LIN {X 0,Y 150.049,Z 459.61,A -85,B 0,C 180,E1 -27742.355,E2 -27742.355} C_VEL
LIN {X 0,Y 146.162,Z 497.421,A -85,B 0,C 180,E1 -27743.604,E2 -27743.604} C_VEL
LIN {X 0,Y 143.307,Z 511.831,A -85,B 0,C 180,E1 -27744.296,E2 -27744.296} C_VEL
LIN {X 0,Y 139.411,Z 525.465,A -85,B 0,C 180,E1 -27745.274,E2 -27745.274} C_VEL
LIN {X 0,Y 134.664,Z 538.406,A -85,B 0,C 180,E1 -27746.652,E2 -27746.652} C_VEL
LIN {X 0,Y 128.857,Z 550.964,A -85,B 0,C 180,E1 -27748.42,E2 -27748.42} C_VEL
LIN {X 0,Y 122.535,Z 562.435,A -85,B 0,C 180,E1 -27750.646,E2 -27750.646} C_VEL
LIN {X 0,Y 115.9,Z 572.988,A -85,B 0,C 180,E1 -27753.511,E2 -27753.511} C_VEL
LIN {X 0,Y 109.403,Z 581.813,A -85,B 0,C 180,E1 -27756.583,E2 -27756.583} C_VEL
LIN {X 0,Y 102.065,Z 590.715,A -85,B 0,C 180,E1 -27760.761,E2 -27760.761} C_VEL
LIN {X 0,Y 94.497,Z 599.259,A -85,B 0,C 180,E1 -27766.532,E2 -27766.532} C_VEL
LIN {X 0,Y 87.771,Z 606.36,A -85,B 0,C 180,E1 -27773.45,E2 -27773.45} C_VEL
LIN {X 0,Y 82.263,Z 612.254,A -85,B 0,C 180,E1 -27781.973,E2 -27781.973} C_VEL
LIN {X 0,Y 79.141,Z 615.759,A -85,B 0,C 180,E1 -27789.193,E2 -27789.193} C_VEL
LIN {X 0,Y 76.993,Z 619.148,A -85,B 0,C 180,E1 -27799.481,E2 -27799.481} C_VEL
LIN {X 0,Y 76.773,Z 621.111,A -85,B 0,C 180,E1 -27810,E2 -27810} C_VEL
LIN {X 0,Y 76.692,Z 621.557,A -85,B 0,C 180,E1 -27815.258,E2 -27815.258} C_VEL
LIN {X 0,Y 77.909,Z 621.446,A -85,B 0,C 180,E1 -27825.702,E2 -27825.702} C_VEL
LIN {X 0,Y 81.239,Z 620.015,A -85,B 0,C 180,E1 -27835.63,E2 -27835.63} C_VEL
LIN {X 0,Y 86.758,Z 617.241,A -85,B 0,C 180,E1 -27844.545,E2 -27844.545} C_VEL
LIN {X 0,Y 94.007,Z 613.047,A -85,B 0,C 180,E1 -27852.287,E2 -27852.287} C_VEL
LIN {X 0,Y 102.811,Z 607.313,A -85,B 0,C 180,E1 -27858.76,E2 -27858.76} C_VEL
LIN {X 0,Y 111.433,Z 600.872,A -85,B 0,C 180,E1 -27863.527,E2 -27863.527} C_VEL
LIN {X 0,Y 120.813,Z 592.893,A -85,B 0,C 180,E1 -27867.513,E2 -27867.513} C_VEL
LIN {X 0,Y 129.752,Z 583.984,A -85,B 0,C 180,E1 -27870.681,E2 -27870.681} C_VEL
LIN {X 0,Y 137.838,Z 574.549,A -85,B 0,C 180,E1 -27873.162,E2 -27873.162} C_VEL
LIN {X 0,Y 146.077,Z 563.405,A -85,B 0,C 180,E1 -27875.246,E2 -27875.246} C_VEL
LIN {X 0,Y 153.73,Z 550.921,A -85,B 0,C 180,E1 -27876.934,E2 -27876.934} C_VEL
LIN {X 0,Y 159.95,Z 538.627,A -85,B 0,C 180,E1 -27878.12,E2 -27878.12} C_VEL
LIN {X 0,Y 161.993,Z 533.397,A -85,B 0,C 180,E1 -27878.765,E2 -27878.765} C_VEL
LIN {X 0,Y 164.34,Z 524.755,A -85,B 0,C 180,E1 -27880.308,E2 -27880.308} C_VEL
LIN {X 0,Y 166.376,Z 515.938,A -85,B 0,C 180,E1 -27881.701,E2 -27881.701} C_VEL
LIN {X 0,Y 167.725,Z 510.353,A -85,B 0,C 180,E1 -27882.131,E2 -27882.131} C_VEL
LIN {X 0,Y 170.729,Z 495.859,A -85,B 0,C 180,E1 -27882.599,E2 -27882.599} C_VEL
LIN {X 0,Y 172.205,Z 483.537,A -85,B 0,C 180,E1 -27882.95,E2 -27882.95} C_VEL
LIN {X 0,Y 171.335,Z 480.194,A -85,B 0,C 180,E1 -27884.69,E2 -27884.69} C_VEL
LIN {X 0,Y 170.04,Z 476.888,A -85,B 0,C 180,E1 -27887.468,E2 -27887.468} C_VEL
LIN {X 0,Y 169.39,Z 475.135,A -85,B 0,C 180,E1 -27889.24,E2 -27889.24} C_VEL
LIN {X 0,Y 168.394,Z 472.197,A -85,B 0,C 180,E1 -27893.298,E2 -27893.298} C_VEL
LIN {X 0,Y 167.964,Z 471.571,A -85,B 0,C 180,E1 -27897.603,E2 -27897.603} C_VEL
LIN {X 0,Y 168.203,Z 471.94,A -85,B 0,C 180,E1 -27901.025,E2 -27901.025} C_VEL
LIN {X 0,Y 168.548,Z 472.677,A -85,B 0,C 180,E1 -27902.988,E2 -27902.988} C_VEL
LIN {X 0,Y 169.83,Z 476.312,A -85,B 0,C 180,E1 -27907.431,E2 -27907.431} C_VEL
LIN {X 0,Y 171.551,Z 480.72,A -85,B 0,C 180,E1 -27911.147,E2 -27911.147} C_VEL
LIN {X 0,Y 172.279,Z 482.684,A -85,B 0,C 180,E1 -27912.442,E2 -27912.442} C_VEL
LIN {X 0,Y 170.181,Z 498.122,A -85,B 0,C 180,E1 -27912.948,E2 -27912.948} C_VEL
LIN {X 0,Y 166.876,Z 512.308,A -85,B 0,C 180,E1 -27913.531,E2 -27913.531} C_VEL
LIN {X 0,Y 162.304,Z 526.088,A -85,B 0,C 180,E1 -27914.331,E2 -27914.331} C_VEL
LIN {X 0,Y 156.664,Z 539.002,A -85,B 0,C 180,E1 -27915.311,E2 -27915.311} C_VEL
LIN {X 0,Y 150.651,Z 550.255,A -85,B 0,C 180,E1 -27916.507,E2 -27916.507} C_VEL
LIN {X 0,Y 143.313,Z 561.692,A -85,B 0,C 180,E1 -27918.167,E2 -27918.167} C_VEL
LIN {X 0,Y 136.335,Z 570.854,A -85,B 0,C 180,E1 -27919.816,E2 -27919.816} C_VEL
LIN {X 0,Y 127.48,Z 580.849,A -85,B 0,C 180,E1 -27922.356,E2 -27922.356} C_VEL
LIN {X 0,Y 118.657,Z 589.402,A -85,B 0,C 180,E1 -27925.41,E2 -27925.41} C_VEL
LIN {X 0,Y 108.853,Z 597.403,A -85,B 0,C 180,E1 -27929.352,E2 -27929.352} C_VEL
LIN {X 0,Y 100.98,Z 603.016,A -85,B 0,C 180,E1 -27933.365,E2 -27933.365} C_VEL
LIN {X 0,Y 91.4,Z 608.87,A -85,B 0,C 180,E1 -27939.741,E2 -27939.741} C_VEL
LIN {X 0,Y 83.132,Z 613.133,A -85,B 0,C 180,E1 -27947.442,E2 -27947.442} C_VEL
LIN {X 0,Y 76.589,Z 615.934,A -85,B 0,C 180,E1 -27956.593,E2 -27956.593} C_VEL
LIN {X 0,Y 71.96,Z 617.365,A -85,B 0,C 180,E1 -27967.004,E2 -27967.004} C_VEL
LIN {X 0,Y 69.801,Z 617.46,A -85,B 0,C 180,E1 -27978.382,E2 -27978.382} C_VEL
LIN {X 0,Y 69.537,Z 617.015,A -85,B 0,C 180,E1 -27984.199,E2 -27984.199} C_VEL
LIN {X 0,Y 69.738,Z 616.244,A -85,B 0,C 180,E1 -27990,E2 -27990} C_VEL
LIN {X 0,Y 71.523,Z 613.704,A -85,B 0,C 180,E1 -28001.334,E2 -28001.334} C_VEL
LIN {X 0,Y 75.408,Z 609.746,A -85,B 0,C 180,E1 -28011.888,E2 -28011.888} C_VEL
LIN {X 0,Y 79.65,Z 605.789,A -85,B 0,C 180,E1 -28019.032,E2 -28019.032} C_VEL
LIN {X 0,Y 84.807,Z 600.885,A -85,B 0,C 180,E1 -28025.457,E2 -28025.457} C_VEL
LIN {X 0,Y 91.913,Z 593.855,A -85,B 0,C 180,E1 -28031.994,E2 -28031.994} C_VEL
LIN {X 0,Y 100.238,Z 585.136,A -85,B 0,C 180,E1 -28037.408,E2 -28037.408} C_VEL
LIN {X 0,Y 107.803,Z 576.023,A -85,B 0,C 180,E1 -28041.473,E2 -28041.473} C_VEL
LIN {X 0,Y 114.35,Z 566.946,A -85,B 0,C 180,E1 -28044.524,E2 -28044.524} C_VEL
LIN {X 0,Y 117.715,Z 561.787,A -85,B 0,C 180,E1 -28045.933,E2 -28045.933} C_VEL
LIN {X 0,Y 124.085,Z 551.102,A -85,B 0,C 180,E1 -28048.166,E2 -28048.166} C_VEL
LIN {X 0,Y 129.839,Z 539.597,A -85,B 0,C 180,E1 -28050.004,E2 -28050.004} C_VEL
LIN {X 0,Y 135.017,Z 527.082,A -85,B 0,C 180,E1 -28051.449,E2 -28051.449} C_VEL
LIN {X 0,Y 139.45,Z 513.144,A -85,B 0,C 180,E1 -28052.656,E2 -28052.656} C_VEL
LIN {X 0,Y 142.659,Z 498.796,A -85,B 0,C 180,E1 -28053.543,E2 -28053.543} C_VEL
LIN {X 0,Y 144.739,Z 483.544,A -85,B 0,C 180,E1 -28054.101,E2 -28054.101} C_VEL
LIN {X 0,Y 146.95,Z 461.559,A -85,B 0,C 180,E1 -28054.774,E2 -28054.774} C_VEL
LIN {X 0,Y 144.028,Z 454.359,A -85,B 0,C 180,E1 -28058.856,E2 -28058.856} C_VEL
LIN {X 0,Y 141.654,Z 449.066,A -85,B 0,C 180,E1 -28063.029,E2 -28063.029} C_VEL
LIN {X 0,Y 139.899,Z 445.503,A -85,B 0,C 180,E1 -28067.182,E2 -28067.182} C_VEL
LIN {X 0,Y 138.613,Z 442.08,A -85,B 0,C 180,E1 -28072.599,E2 -28072.599} C_VEL
LIN {X 0,Y 138.35,Z 441.632,A -85,B 0,C 180,E1 -28079.999,E2 -28079.999} C_VEL
LIN {X 0,Y 138.739,Z 442.236,A -85,B 0,C 180,E1 -28082.721,E2 -28082.721} C_VEL
LIN {X 0,Y 140.479,Z 446.546,A -85,B 0,C 180,E1 -28088.969,E2 -28088.969} C_VEL
LIN {X 0,Y 142.08,Z 450.095,A -85,B 0,C 180,E1 -28092.467,E2 -28092.467} C_VEL
LIN {X 0,Y 144.231,Z 454.8,A -85,B 0,C 180,E1 -28096.089,E2 -28096.089} C_VEL
LIN {X 0,Y 146.279,Z 459.975,A -85,B 0,C 180,E1 -28099.014,E2 -28099.014} C_VEL
LIN {X 0,Y 146.933,Z 462.506,A -85,B 0,C 180,E1 -28099.966,E2 -28099.966} C_VEL
LIN {X 0,Y 143.315,Z 496.479,A -85,B 0,C 180,E1 -28101.022,E2 -28101.022} C_VEL
LIN {X 0,Y 140.517,Z 510.666,A -85,B 0,C 180,E1 -28101.661,E2 -28101.661} C_VEL
LIN {X 0,Y 136.534,Z 524.499,A -85,B 0,C 180,E1 -28102.583,E2 -28102.583} C_VEL
LIN {X 0,Y 131.61,Z 537.6,A -85,B 0,C 180,E1 -28103.868,E2 -28103.868} C_VEL
LIN {X 0,Y 125.623,Z 550.277,A -85,B 0,C 180,E1 -28105.562,E2 -28105.562} C_VEL
LIN {X 0,Y 119.038,Z 561.83,A -85,B 0,C 180,E1 -28107.675,E2 -28107.675} C_VEL
LIN {X 0,Y 112.115,Z 572.453,A -85,B 0,C 180,E1 -28110.466,E2 -28110.466} C_VEL
LIN {X 0,Y 105.302,Z 581.333,A -85,B 0,C 180,E1 -28113.46,E2 -28113.46} C_VEL
LIN {X 0,Y 97.542,Z 590.281,A -85,B 0,C 180,E1 -28117.574,E2 -28117.574} C_VEL
LIN {X 0,Y 89.44,Z 598.865,A -85,B 0,C 180,E1 -28123.377,E2 -28123.377} C_VEL
LIN {X 0,Y 82.455,Z 605.679,A -85,B 0,C 180,E1 -28130.093,E2 -28130.093} C_VEL
LIN {X 0,Y 77.412,Z 610.54,A -85,B 0,C 180,E1 -28136.994,E2 -28136.994} C_VEL
LIN {X 0,Y 72.497,Z 615.465,A -85,B 0,C 180,E1 -28147.185,E2 -28147.185} C_VEL
LIN {X 0,Y 69.998,Z 618.884,A -85,B 0,C 180,E1 -28158.416,E2 -28158.416} C_VEL
LIN {X 0,Y 69.668,Z 620.882,A -85,B 0,C 180,E1 -28170,E2 -28170} C_VEL
LIN {X 0,Y 70.04,Z 621.47,A -85,B 0,C 180,E1 -28181.577,E2 -28181.577} C_VEL
LIN {X 0,Y 72.635,Z 620.726,A -85,B 0,C 180,E1 -28192.77,E2 -28192.77} C_VEL
LIN {X 0,Y 77.698,Z 618.659,A -85,B 0,C 180,E1 -28202.869,E2 -28202.869} C_VEL
LIN {X 0,Y 84.864,Z 615.106,A -85,B 0,C 180,E1 -28211.814,E2 -28211.814} C_VEL
LIN {X 0,Y 93.403,Z 610.3,A -85,B 0,C 180,E1 -28218.803,E2 -28218.803} C_VEL
LIN {X 0,Y 103.353,Z 603.767,A -85,B 0,C 180,E1 -28224.687,E2 -28224.687} C_VEL
LIN {X 0,Y 112.871,Z 596.52,A -85,B 0,C 180,E1 -28228.888,E2 -28228.888} C_VEL
LIN {X 0,Y 122.901,Z 587.576,A -85,B 0,C 180,E1 -28232.419,E2 -28232.419} C_VEL
LIN {X 0,Y 131.772,Z 578.207,A -85,B 0,C 180,E1 -28235.052,E2 -28235.052} C_VEL
LIN {X 0,Y 140.158,Z 567.852,A -85,B 0,C 180,E1 -28237.131,E2 -28237.131} C_VEL
LIN {X 0,Y 147.936,Z 556.453,A -85,B 0,C 180,E1 -28238.801,E2 -28238.801} C_VEL
LIN {X 0,Y 155.083,Z 543.84,A -85,B 0,C 180,E1 -28240.11,E2 -28240.11} C_VEL
LIN {X 0,Y 160.72,Z 531.595,A -85,B 0,C 180,E1 -28241.02,E2 -28241.02} C_VEL
LIN {X 0,Y 164.981,Z 519.887,A -85,B 0,C 180,E1 -28241.707,E2 -28241.707} C_VEL
LIN {X 0,Y 167.725,Z 510.353,A -85,B 0,C 180,E1 -28242.131,E2 -28242.131} C_VEL
LIN {X 0,Y 168.511,Z 506.584,A -85,B 0,C 180,E1 -28242.467,E2 -28242.467} C_VEL
LIN {X 0,Y 169.026,Z 500.717,A -85,B 0,C 180,E1 -28243.582,E2 -28243.582} C_VEL
LIN {X 0,Y 169.343,Z 494.798,A -85,B 0,C 180,E1 -28244.697,E2 -28244.697} C_VEL
LIN {X 0,Y 169.698,Z 490.936,A -85,B 0,C 180,E1 -28245.028,E2 -28245.028} C_VEL
LIN {X 0,Y 170.124,Z 487.442,A -85,B 0,C 180,E1 -28245.128,E2 -28245.128} C_VEL
LIN {X 0,Y 169.207,Z 484.494,A -85,B 0,C 180,E1 -28247.253,E2 -28247.253} C_VEL
LIN {X 0,Y 168.169,Z 481.676,A -85,B 0,C 180,E1 -28250.226,E2 -28250.226} C_VEL
LIN {X 0,Y 167.507,Z 479.256,A -85,B 0,C 180,E1 -28253.375,E2 -28253.375} C_VEL
LIN {X 0,Y 167.101,Z 478.601,A -85,B 0,C 180,E1 -28257.59,E2 -28257.59} C_VEL
LIN {X 0,Y 167.358,Z 479.058,A -85,B 0,C 180,E1 -28261.204,E2 -28261.204} C_VEL
LIN {X 0,Y 167.602,Z 479.736,A -85,B 0,C 180,E1 -28262.705,E2 -28262.705} C_VEL
LIN {X 0,Y 168.604,Z 482.861,A -85,B 0,C 180,E1 -28266.583,E2 -28266.583} C_VEL
LIN {X 0,Y 169.946,Z 486.698,A -85,B 0,C 180,E1 -28269.898,E2 -28269.898} C_VEL
LIN {X 0,Y 170.129,Z 487.262,A -85,B 0,C 180,E1 -28270.307,E2 -28270.307} C_VEL
LIN {X 0,Y 167.681,Z 501.969,A -85,B 0,C 180,E1 -28270.745,E2 -28270.745} C_VEL
LIN {X 0,Y 164.24,Z 515.205,A -85,B 0,C 180,E1 -28271.311,E2 -28271.311} C_VEL
LIN {X 0,Y 159.041,Z 529.586,A -85,B 0,C 180,E1 -28272.121,E2 -28272.121} C_VEL
LIN {X 0,Y 153.291,Z 541.822,A -85,B 0,C 180,E1 -28273.027,E2 -28273.027} C_VEL
LIN {X 0,Y 146.36,Z 553.9,A -85,B 0,C 180,E1 -28274.337,E2 -28274.337} C_VEL
LIN {X 0,Y 138.842,Z 564.736,A -85,B 0,C 180,E1 -28275.895,E2 -28275.895} C_VEL
LIN {X 0,Y 130.933,Z 574.323,A -85,B 0,C 180,E1 -28277.68,E2 -28277.68} C_VEL
LIN {X 0,Y 121.319,Z 584.303,A -85,B 0,C 180,E1 -28280.341,E2 -28280.341} C_VEL
LIN {X 0,Y 111.318,Z 593.061,A -85,B 0,C 180,E1 -28283.73,E2 -28283.73} C_VEL
LIN {X 0,Y 102.691,Z 599.44,A -85,B 0,C 180,E1 -28287.163,E2 -28287.163} C_VEL
LIN {X 0,Y 93.87,Z 605.087,A -85,B 0,C 180,E1 -28291.608,E2 -28291.608} C_VEL
LIN {X 0,Y 84.584,Z 610.198,A -85,B 0,C 180,E1 -28297.874,E2 -28297.874} C_VEL
LIN {X 0,Y 77.98,Z 613.256,A -85,B 0,C 180,E1 -28303.862,E2 -28303.862} C_VEL
LIN {X 0,Y 70.698,Z 616.087,A -85,B 0,C 180,E1 -28313.383,E2 -28313.383} C_VEL
LIN {X 0,Y 65.424,Z 617.546,A -85,B 0,C 180,E1 -28324.552,E2 -28324.552} C_VEL
LIN {X 0,Y 62.814,Z 617.67,A -85,B 0,C 180,E1 -28337.069,E2 -28337.069} C_VEL
LIN {X 0,Y 62.444,Z 617.239,A -85,B 0,C 180,E1 -28343.537,E2 -28343.537} C_VEL
LIN {X 0,Y 62.63,Z 616.481,A -85,B 0,C 180,E1 -28350,E2 -28350} C_VEL
LIN {X 0,Y 64.601,Z 613.976,A -85,B 0,C 180,E1 -28362.567,E2 -28362.567} C_VEL
LIN {X 0,Y 68.888,Z 610.058,A -85,B 0,C 180,E1 -28374.084,E2 -28374.084} C_VEL
LIN {X 0,Y 75.305,Z 604.6,A -85,B 0,C 180,E1 -28384.053,E2 -28384.053} C_VEL
LIN {X 0,Y 81.202,Z 599.439,A -85,B 0,C 180,E1 -28390.475,E2 -28390.475} C_VEL
LIN {X 0,Y 89.222,Z 591.981,A -85,B 0,C 180,E1 -28396.771,E2 -28396.771} C_VEL
LIN {X 0,Y 96.88,Z 584.207,A -85,B 0,C 180,E1 -28401.246,E2 -28401.246} C_VEL
LIN {X 0,Y 104.933,Z 574.836,A -85,B 0,C 180,E1 -28405.131,E2 -28405.131} C_VEL
LIN {X 0,Y 113.242,Z 563.424,A -85,B 0,C 180,E1 -28408.578,E2 -28408.578} C_VEL
LIN {X 0,Y 116.829,Z 557.892,A -85,B 0,C 180,E1 -28409.855,E2 -28409.855} C_VEL
LIN {X 0,Y 123.513,Z 546.338,A -85,B 0,C 180,E1 -28411.881,E2 -28411.881} C_VEL
LIN {X 0,Y 128.74,Z 535.41,A -85,B 0,C 180,E1 -28413.371,E2 -28413.371} C_VEL
LIN {X 0,Y 134.076,Z 521.62,A -85,B 0,C 180,E1 -28414.718,E2 -28414.718} C_VEL
LIN {X 0,Y 138.049,Z 507.765,A -85,B 0,C 180,E1 -28415.728,E2 -28415.728} C_VEL
LIN {X 0,Y 140.871,Z 493.399,A -85,B 0,C 180,E1 -28416.432,E2 -28416.432} C_VEL
LIN {X 0,Y 144.022,Z 465.257,A -85,B 0,C 180,E1 -28417.245,E2 -28417.245} C_VEL
LIN {X 0,Y 141.854,Z 459.58,A -85,B 0,C 180,E1 -28420.766,E2 -28420.766} C_VEL
LIN {X 0,Y 139.995,Z 455.172,A -85,B 0,C 180,E1 -28424.531,E2 -28424.531} C_VEL
LIN {X 0,Y 138.818,Z 452.412,A -85,B 0,C 180,E1 -28427.699,E2 -28427.699} C_VEL
LIN {X 0,Y 137.66,Z 449.081,A -85,B 0,C 180,E1 -28433.079,E2 -28433.079} C_VEL
LIN {X 0,Y 137.482,Z 448.688,A -85,B 0,C 180,E1 -28439.999,E2 -28439.999} C_VEL
LIN {X 0,Y 137.764,Z 449.206,A -85,B 0,C 180,E1 -28442.192,E2 -28442.192} C_VEL
LIN {X 0,Y 139.24,Z 453.304,A -85,B 0,C 180,E1 -28448.16,E2 -28448.16} C_VEL
LIN {X 0,Y 140.694,Z 456.807,A -85,B 0,C 180,E1 -28451.643,E2 -28451.643} C_VEL
LIN {X 0,Y 142.737,Z 461.782,A -85,B 0,C 180,E1 -28455.38,E2 -28455.38} C_VEL
LIN {X 0,Y 144.045,Z 465.45,A -85,B 0,C 180,E1 -28457.445,E2 -28457.445} C_VEL
LIN {X 0,Y 140.533,Z 496.919,A -85,B 0,C 180,E1 -28458.392,E2 -28458.392} C_VEL
LIN {X 0,Y 137.596,Z 511.158,A -85,B 0,C 180,E1 -28459.003,E2 -28459.003} C_VEL
LIN {X 0,Y 133.165,Z 525.797,A -85,B 0,C 180,E1 -28459.933,E2 -28459.933} C_VEL
LIN {X 0,Y 128.113,Z 538.574,A -85,B 0,C 180,E1 -28461.158,E2 -28461.158} C_VEL
LIN {X 0,Y 121.945,Z 551.024,A -85,B 0,C 180,E1 -28462.761,E2 -28462.761} C_VEL
LIN {X 0,Y 115.07,Z 562.528,A -85,B 0,C 180,E1 -28464.805,E2 -28464.805} C_VEL
LIN {X 0,Y 107.227,Z 573.872,A -85,B 0,C 180,E1 -28467.768,E2 -28467.768} C_VEL
LIN {X 0,Y 98.762,Z 584.063,A -85,B 0,C 180,E1 -28471.357,E2 -28471.357} C_VEL
LIN {X 0,Y 90.781,Z 592.521,A -85,B 0,C 180,E1 -28475.622,E2 -28475.622} C_VEL
LIN {X 0,Y 82.369,Z 600.609,A -85,B 0,C 180,E1 -28481.705,E2 -28481.705} C_VEL
LIN {X 0,Y 75.044,Z 607.12,A -85,B 0,C 180,E1 -28489.037,E2 -28489.037} C_VEL
LIN {X 0,Y 68.476,Z 612.893,A -85,B 0,C 180,E1 -28499.125,E2 -28499.125} C_VEL
LIN {X 0,Y 64.166,Z 617.078,A -85,B 0,C 180,E1 -28510.817,E2 -28510.817} C_VEL
LIN {X 0,Y 62.506,Z 619.809,A -85,B 0,C 180,E1 -28523.544,E2 -28523.544} C_VEL
LIN {X 0,Y 62.558,Z 620.65,A -85,B 0,C 180,E1 -28530,E2 -28530} C_VEL
LIN {X 0,Y 62.534,Z 621.128,A -85,B 0,C 180,E1 -28536.453,E2 -28536.453} C_VEL
LIN {X 0,Y 64.277,Z 621.078,A -85,B 0,C 180,E1 -28549.149,E2 -28549.149} C_VEL
LIN {X 0,Y 68.665,Z 619.705,A -85,B 0,C 180,E1 -28560.782,E2 -28560.782} C_VEL
LIN {X 0,Y 75.423,Z 616.988,A -85,B 0,C 180,E1 -28570.713,E2 -28570.713} C_VEL
LIN {X 0,Y 83.985,Z 612.852,A -85,B 0,C 180,E1 -28578.863,E2 -28578.863} C_VEL
LIN {X 0,Y 94.008,Z 607.181,A -85,B 0,C 180,E1 -28585.322,E2 -28585.322} C_VEL
LIN {X 0,Y 103.59,Z 600.81,A -85,B 0,C 180,E1 -28589.885,E2 -28589.885} C_VEL
LIN {X 0,Y 113.796,Z 592.908,A -85,B 0,C 180,E1 -28593.576,E2 -28593.576} C_VEL
LIN {X 0,Y 124.009,Z 583.495,A -85,B 0,C 180,E1 -28596.628,E2 -28596.628} C_VEL
LIN {X 0,Y 132.037,Z 574.754,A -85,B 0,C 180,E1 -28598.668,E2 -28598.668} C_VEL
LIN {X 0,Y 140.73,Z 563.75,A -85,B 0,C 180,E1 -28600.497,E2 -28600.497} C_VEL
LIN {X 0,Y 148.759,Z 551.494,A -85,B 0,C 180,E1 -28601.952,E2 -28601.952} C_VEL
LIN {X 0,Y 155.268,Z 539.357,A -85,B 0,C 180,E1 -28602.98,E2 -28602.98} C_VEL
LIN {X 0,Y 160.985,Z 525.903,A -85,B 0,C 180,E1 -28603.831,E2 -28603.831} C_VEL
LIN {X 0,Y 165.497,Z 511.915,A -85,B 0,C 180,E1 -28604.434,E2 -28604.434} C_VEL
LIN {X 0,Y 168.659,Z 497.752,A -85,B 0,C 180,E1 -28604.87,E2 -28604.87} C_VEL
LIN {X 0,Y 169.698,Z 490.936,A -85,B 0,C 180,E1 -28605.028,E2 -28605.028} C_VEL
LIN {X 0,Y 169.759,Z 489.264,A -85,B 0,C 180,E1 -28605.314,E2 -28605.314} C_VEL
LIN {X 0,Y 169.505,Z 487.892,A -85,B 0,C 180,E1 -28606.039,E2 -28606.039} C_VEL
LIN {X 0,Y 168.884,Z 487.154,A -85,B 0,C 180,E1 -28607.303,E2 -28607.303} C_VEL
LIN {X 0,Y 167.021,Z 487.859,A -85,B 0,C 180,E1 -28611.303,E2 -28611.303} C_VEL
LIN {X 0,Y 166.803,Z 487.549,A -85,B 0,C 180,E1 -28612.126,E2 -28612.126} C_VEL
LIN {X 0,Y 166.535,Z 486.182,A -85,B 0,C 180,E1 -28613.945,E2 -28613.945} C_VEL
LIN {X 0,Y 166.233,Z 485.659,A -85,B 0,C 180,E1 -28617.578,E2 -28617.578} C_VEL
LIN {X 0,Y 166.489,Z 486.126,A -85,B 0,C 180,E1 -28621.21,E2 -28621.21} C_VEL
LIN {X 0,Y 166.752,Z 487.282,A -85,B 0,C 180,E1 -28623.021,E2 -28623.021} C_VEL
LIN {X 0,Y 167.441,Z 489.702,A -85,B 0,C 180,E1 -28626.024,E2 -28626.024} C_VEL
LIN {X 0,Y 168.082,Z 491.892,A -85,B 0,C 180,E1 -28628.037,E2 -28628.037} C_VEL
LIN {X 0,Y 165.362,Z 505.861,A -85,B 0,C 180,E1 -28628.485,E2 -28628.485} C_VEL
LIN {X 0,Y 161.46,Z 519.273,A -85,B 0,C 180,E1 -28629.069,E2 -28629.069} C_VEL
LIN {X 0,Y 156.022,Z 532.967,A -85,B 0,C 180,E1 -28629.815,E2 -28629.815} C_VEL
LIN {X 0,Y 149.407,Z 545.93,A -85,B 0,C 180,E1 -28630.785,E2 -28630.785} C_VEL
LIN {X 0,Y 141.958,Z 557.838,A -85,B 0,C 180,E1 -28632.101,E2 -28632.101} C_VEL
LIN {X 0,Y 133.79,Z 568.618,A -85,B 0,C 180,E1 -28633.636,E2 -28633.636} C_VEL
LIN {X 0,Y 124.14,Z 579.267,A -85,B 0,C 180,E1 -28635.753,E2 -28635.753} C_VEL
LIN {X 0,Y 114.744,Z 588.05,A -85,B 0,C 180,E1 -28638.343,E2 -28638.343} C_VEL
LIN {X 0,Y 104.074,Z 596.417,A -85,B 0,C 180,E1 -28641.793,E2 -28641.793} C_VEL
LIN {X 0,Y 93.842,Z 603.128,A -85,B 0,C 180,E1 -28646.011,E2 -28646.011} C_VEL
LIN {X 0,Y 85.542,Z 607.724,A -85,B 0,C 180,E1 -28650.382,E2 -28650.382} C_VEL
LIN {X 0,Y 77.862,Z 611.408,A -85,B 0,C 180,E1 -28655.672,E2 -28655.672} C_VEL
LIN {X 0,Y 68.901,Z 614.986,A -85,B 0,C 180,E1 -28664.438,E2 -28664.438} C_VEL
LIN {X 0,Y 61.731,Z 617.152,A -85,B 0,C 180,E1 -28675.302,E2 -28675.302} C_VEL
LIN {X 0,Y 57.053,Z 617.97,A -85,B 0,C 180,E1 -28688.312,E2 -28688.312} C_VEL
LIN {X 0,Y 55.357,Z 617.463,A -85,B 0,C 180,E1 -28702.706,E2 -28702.706} C_VEL
LIN {X 0,Y 55.516,Z 616.719,A -85,B 0,C 180,E1 -28710,E2 -28710} C_VEL
LIN {X 0,Y 57.714,Z 614.244,A -85,B 0,C 180,E1 -28724.096,E2 -28724.096} C_VEL
LIN {X 0,Y 62.493,Z 610.37,A -85,B 0,C 180,E1 -28736.734,E2 -28736.734} C_VEL
LIN {X 0,Y 67.621,Z 606.445,A -85,B 0,C 180,E1 -28744.864,E2 -28744.864} C_VEL
LIN {X 0,Y 75.967,Z 599.812,A -85,B 0,C 180,E1 -28753.936,E2 -28753.936} C_VEL
LIN {X 0,Y 84.541,Z 592.4,A -85,B 0,C 180,E1 -28760.261,E2 -28760.261} C_VEL
LIN {X 0,Y 92.617,Z 584.666,A -85,B 0,C 180,E1 -28764.66,E2 -28764.66} C_VEL
LIN {X 0,Y 101.061,Z 575.351,A -85,B 0,C 180,E1 -28768.418,E2 -28768.418} C_VEL
LIN {X 0,Y 109.727,Z 564.001,A -85,B 0,C 180,E1 -28771.726,E2 -28771.726} C_VEL
LIN {X 0,Y 113.447,Z 558.506,A -85,B 0,C 180,E1 -28772.939,E2 -28772.939} C_VEL
LIN {X 0,Y 120.35,Z 547.039,A -85,B 0,C 180,E1 -28774.843,E2 -28774.843} C_VEL
LIN {X 0,Y 125.737,Z 536.23,A -85,B 0,C 180,E1 -28776.245,E2 -28776.245} C_VEL
LIN {X 0,Y 131.2,Z 522.675,A -85,B 0,C 180,E1 -28777.496,E2 -28777.496} C_VEL
LIN {X 0,Y 135.39,Z 508.746,A -85,B 0,C 180,E1 -28778.453,E2 -28778.453} C_VEL
LIN {X 0,Y 138.287,Z 494.741,A -85,B 0,C 180,E1 -28779.126,E2 -28779.126} C_VEL
LIN {X 0,Y 141.32,Z 468.998,A -85,B 0,C 180,E1 -28779.869,E2 -28779.869} C_VEL
LIN {X 0,Y 139.577,Z 464.13,A -85,B 0,C 180,E1 -28783.3,E2 -28783.3} C_VEL
LIN {X 0,Y 138.326,Z 460.973,A -85,B 0,C 180,E1 -28786.379,E2 -28786.379} C_VEL
LIN {X 0,Y 137.545,Z 458.947,A -85,B 0,C 180,E1 -28788.906,E2 -28788.906} C_VEL
LIN {X 0,Y 136.728,Z 456.16,A -85,B 0,C 180,E1 -28793.432,E2 -28793.432} C_VEL
LIN {X 0,Y 136.472,Z 455.714,A -85,B 0,C 180,E1 -28797.047,E2 -28797.047} C_VEL
LIN {X 0,Y 136.78,Z 455.964,A -85,B 0,C 180,E1 -28801.379,E2 -28801.379} C_VEL
LIN {X 0,Y 138.071,Z 460.115,A -85,B 0,C 180,E1 -28807.448,E2 -28807.448} C_VEL
LIN {X 0,Y 139.483,Z 463.842,A -85,B 0,C 180,E1 -28811.12,E2 -28811.12} C_VEL
LIN {X 0,Y 141.374,Z 469.056,A -85,B 0,C 180,E1 -28814.847,E2 -28814.847} C_VEL
LIN {X 0,Y 138.122,Z 496.971,A -85,B 0,C 180,E1 -28815.649,E2 -28815.649} C_VEL
LIN {X 0,Y 134.96,Z 511.708,A -85,B 0,C 180,E1 -28816.236,E2 -28816.236} C_VEL
LIN {X 0,Y 130.507,Z 525.949,A -85,B 0,C 180,E1 -28817.085,E2 -28817.085} C_VEL
LIN {X 0,Y 125.718,Z 537.761,A -85,B 0,C 180,E1 -28818.13,E2 -28818.13} C_VEL
LIN {X 0,Y 119.377,Z 550.332,A -85,B 0,C 180,E1 -28819.616,E2 -28819.616} C_VEL
LIN {X 0,Y 112.324,Z 561.798,A -85,B 0,C 180,E1 -28821.454,E2 -28821.454} C_VEL
LIN {X 0,Y 104.779,Z 572.431,A -85,B 0,C 180,E1 -28824.034,E2 -28824.034} C_VEL
LIN {X 0,Y 96.694,Z 582.012,A -85,B 0,C 180,E1 -28827.08,E2 -28827.08} C_VEL
LIN {X 0,Y 88.155,Z 590.779,A -85,B 0,C 180,E1 -28831.016,E2 -28831.016} C_VEL
LIN {X 0,Y 79.025,Z 599.202,A -85,B 0,C 180,E1 -28836.831,E2 -28836.831} C_VEL
LIN {X 0,Y 70.918,Z 605.898,A -85,B 0,C 180,E1 -28843.922,E2 -28843.922} C_VEL
LIN {X 0,Y 64.106,Z 611.323,A -85,B 0,C 180,E1 -28852.917,E2 -28852.917} C_VEL
LIN {X 0,Y 59.566,Z 614.878,A -85,B 0,C 180,E1 -28861.84,E2 -28861.84} C_VEL
LIN {X 0,Y 56.1,Z 618.356,A -85,B 0,C 180,E1 -28875.49,E2 -28875.49} C_VEL
LIN {X 0,Y 55.444,Z 619.559,A -85,B 0,C 180,E1 -28882.718,E2 -28882.718} C_VEL
LIN {X 0,Y 55.469,Z 620.415,A -85,B 0,C 180,E1 -28890,E2 -28890} C_VEL
LIN {X 0,Y 56.147,Z 621.064,A -85,B 0,C 180,E1 -28904.498,E2 -28904.498} C_VEL
LIN {X 0,Y 59.707,Z 620.382,A -85,B 0,C 180,E1 -28918.089,E2 -28918.089} C_VEL
LIN {X 0,Y 66.126,Z 618.376,A -85,B 0,C 180,E1 -28929.62,E2 -28929.62} C_VEL
LIN {X 0,Y 74.582,Z 614.991,A -85,B 0,C 180,E1 -28938.927,E2 -28938.927} C_VEL
LIN {X 0,Y 84.688,Z 610.138,A -85,B 0,C 180,E1 -28946.087,E2 -28946.087} C_VEL
LIN {X 0,Y 95.813,Z 603.672,A -85,B 0,C 180,E1 -28951.67,E2 -28951.67} C_VEL
LIN {X 0,Y 106.229,Z 596.499,A -85,B 0,C 180,E1 -28955.463,E2 -28955.463} C_VEL
LIN {X 0,Y 116.7,Z 587.916,A -85,B 0,C 180,E1 -28958.513,E2 -28958.513} C_VEL
LIN {X 0,Y 126.429,Z 578.395,A -85,B 0,C 180,E1 -28960.911,E2 -28960.911} C_VEL
LIN {X 0,Y 135.273,Z 568.178,A -85,B 0,C 180,E1 -28962.682,E2 -28962.682} C_VEL
LIN {X 0,Y 143.426,Z 556.939,A -85,B 0,C 180,E1 -28964.08,E2 -28964.08} C_VEL
LIN {X 0,Y 150.858,Z 544.526,A -85,B 0,C 180,E1 -28965.169,E2 -28965.169} C_VEL
LIN {X 0,Y 156.694,Z 532.56,A -85,B 0,C 180,E1 -28965.913,E2 -28965.913} C_VEL
LIN {X 0,Y 161.297,Z 520.677,A -85,B 0,C 180,E1 -28966.507,E2 -28966.507} C_VEL
LIN {X 0,Y 165.363,Z 506.596,A -85,B 0,C 180,E1 -28967.007,E2 -28967.007} C_VEL
LIN {X 0,Y 168.077,Z 492.26,A -85,B 0,C 180,E1 -28967.384,E2 -28967.384} C_VEL
LIN {X 0,Y 168.1,Z 491.778,A -85,B 0,C 180,E1 -28967.474,E2 -28967.474} C_VEL
LIN {X 0,Y 167.135,Z 488.536,A -85,B 0,C 180,E1 -28970.699,E2 -28970.699} C_VEL
LIN {X 0,Y 166.803,Z 487.549,A -85,B 0,C 180,E1 -28972.126,E2 -28972.126} C_VEL
LIN {X 0,Y 166.384,Z 487.125,A -85,B 0,C 180,E1 -28974.149,E2 -28974.149} C_VEL
LIN {X 0,Y 166.017,Z 487.945,A -85,B 0,C 180,E1 -28976.178,E2 -28976.178} C_VEL
LIN {X 0,Y 165.675,Z 490.254,A -85,B 0,C 180,E1 -28978.85,E2 -28978.85} C_VEL
LIN {X 0,Y 165.629,Z 494.408,A -85,B 0,C 180,E1 -28982.852,E2 -28982.852} C_VEL
LIN {X 0,Y 166.067,Z 496.488,A -85,B 0,C 180,E1 -28985.465,E2 -28985.465} C_VEL
LIN {X 0,Y 166.12,Z 496.802,A -85,B 0,C 180,E1 -28985.752,E2 -28985.752} C_VEL
LIN {X 0,Y 162.855,Z 510.864,A -85,B 0,C 180,E1 -28986.211,E2 -28986.211} C_VEL
LIN {X 0,Y 158.501,Z 524.026,A -85,B 0,C 180,E1 -28986.794,E2 -28986.794} C_VEL
LIN {X 0,Y 152.415,Z 537.872,A -85,B 0,C 180,E1 -28987.523,E2 -28987.523} C_VEL
LIN {X 0,Y 146.316,Z 548.878,A -85,B 0,C 180,E1 -28988.325,E2 -28988.325} C_VEL
LIN {X 0,Y 138.127,Z 561.15,A -85,B 0,C 180,E1 -28989.66,E2 -28989.66} C_VEL
LIN {X 0,Y 128.97,Z 572.306,A -85,B 0,C 180,E1 -28991.219,E2 -28991.219} C_VEL
LIN {X 0,Y 119.137,Z 582.306,A -85,B 0,C 180,E1 -28993.255,E2 -28993.255} C_VEL
LIN {X 0,Y 109.52,Z 590.586,A -85,B 0,C 180,E1 -28995.725,E2 -28995.725} C_VEL
LIN {X 0,Y 98.512,Z 598.481,A -85,B 0,C 180,E1 -28999.042,E2 -28999.042} C_VEL
LIN {X 0,Y 87.647,Z 604.966,A -85,B 0,C 180,E1 -29003.346,E2 -29003.346} C_VEL
LIN {X 0,Y 76.582,Z 610.385,A -85,B 0,C 180,E1 -29009.328,E2 -29009.328} C_VEL
LIN {X 0,Y 68.781,Z 613.505,A -85,B 0,C 180,E1 -29015.17,E2 -29015.17} C_VEL
LIN {X 0,Y 59.762,Z 616.394,A -85,B 0,C 180,E1 -29025.121,E2 -29025.121} C_VEL
LIN {X 0,Y 52.825,Z 617.911,A -85,B 0,C 180,E1 -29037.847,E2 -29037.847} C_VEL
LIN {X 0,Y 48.955,Z 618.091,A -85,B 0,C 180,E1 -29053.314,E2 -29053.314} C_VEL
LIN {X 0,Y 48.299,Z 617.687,A -85,B 0,C 180,E1 -29061.633,E2 -29061.633} C_VEL
LIN {X 0,Y 48.393,Z 616.957,A -85,B 0,C 180,E1 -29070,E2 -29070} C_VEL
LIN {X 0,Y 50.866,Z 614.51,A -85,B 0,C 180,E1 -29086.041,E2 -29086.041} C_VEL
LIN {X 0,Y 56.26,Z 610.675,A -85,B 0,C 180,E1 -29099.979,E2 -29099.979} C_VEL
LIN {X 0,Y 64.077,Z 605.287,A -85,B 0,C 180,E1 -29111.154,E2 -29111.154} C_VEL
LIN {X 0,Y 71.033,Z 600.177,A -85,B 0,C 180,E1 -29117.906,E2 -29117.906} C_VEL
LIN {X 0,Y 80.208,Z 592.815,A -85,B 0,C 180,E1 -29124.145,E2 -29124.145} C_VEL
LIN {X 0,Y 88.715,Z 585.114,A -85,B 0,C 180,E1 -29128.388,E2 -29128.388} C_VEL
LIN {X 0,Y 97.539,Z 575.86,A -85,B 0,C 180,E1 -29131.965,E2 -29131.965} C_VEL
LIN {X 0,Y 105.831,Z 565.633,A -85,B 0,C 180,E1 -29134.798,E2 -29134.798} C_VEL
LIN {X 0,Y 109.61,Z 560.291,A -85,B 0,C 180,E1 -29136.02,E2 -29136.02} C_VEL
LIN {X 0,Y 116.728,Z 549.159,A -85,B 0,C 180,E1 -29137.776,E2 -29137.776} C_VEL
LIN {X 0,Y 123.065,Z 537.05,A -85,B 0,C 180,E1 -29139.252,E2 -29139.252} C_VEL
LIN {X 0,Y 128.63,Z 523.761,A -85,B 0,C 180,E1 -29140.397,E2 -29140.397} C_VEL
LIN {X 0,Y 133.113,Z 509.447,A -85,B 0,C 180,E1 -29141.311,E2 -29141.311} C_VEL
LIN {X 0,Y 136.146,Z 495.373,A -85,B 0,C 180,E1 -29141.937,E2 -29141.937} C_VEL
LIN {X 0,Y 138.911,Z 472.937,A -85,B 0,C 180,E1 -29142.575,E2 -29142.575} C_VEL
LIN {X 0,Y 137.513,Z 468.654,A -85,B 0,C 180,E1 -29146.061,E2 -29146.061} C_VEL
LIN {X 0,Y 136.486,Z 465.79,A -85,B 0,C 180,E1 -29149.523,E2 -29149.523} C_VEL
LIN {X 0,Y 135.78,Z 463.103,A -85,B 0,C 180,E1 -29154.057,E2 -29154.057} C_VEL
LIN {X 0,Y 135.746,Z 462.798,A -85,B 0,C 180,E1 -29159.999,E2 -29159.999} C_VEL
LIN {X 0,Y 135.895,Z 463.481,A -85,B 0,C 180,E1 -29161.62,E2 -29161.62} C_VEL
LIN {X 0,Y 136.885,Z 466.801,A -85,B 0,C 180,E1 -29166.587,E2 -29166.587} C_VEL
LIN {X 0,Y 138.198,Z 470.681,A -85,B 0,C 180,E1 -29170.392,E2 -29170.392} C_VEL
LIN {X 0,Y 138.953,Z 472.989,A -85,B 0,C 180,E1 -29172.14,E2 -29172.14} C_VEL
LIN {X 0,Y 135.979,Z 497.351,A -85,B 0,C 180,E1 -29172.823,E2 -29172.823} C_VEL
LIN {X 0,Y 132.751,Z 511.905,A -85,B 0,C 180,E1 -29173.356,E2 -29173.356} C_VEL
LIN {X 0,Y 128.185,Z 526.102,A -85,B 0,C 180,E1 -29174.127,E2 -29174.127} C_VEL
LIN {X 0,Y 122.865,Z 538.722,A -85,B 0,C 180,E1 -29175.144,E2 -29175.144} C_VEL
LIN {X 0,Y 116.36,Z 551.068,A -85,B 0,C 180,E1 -29176.497,E2 -29176.497} C_VEL
LIN {X 0,Y 109.115,Z 562.371,A -85,B 0,C 180,E1 -29178.188,E2 -29178.188} C_VEL
LIN {X 0,Y 100.677,Z 573.648,A -85,B 0,C 180,E1 -29180.819,E2 -29180.819} C_VEL
LIN {X 0,Y 92.141,Z 583.144,A -85,B 0,C 180,E1 -29183.752,E2 -29183.752} C_VEL
LIN {X 0,Y 83.247,Z 591.687,A -85,B 0,C 180,E1 -29187.57,E2 -29187.57} C_VEL
LIN {X 0,Y 73.618,Z 599.855,A -85,B 0,C 180,E1 -29193.349,E2 -29193.349} C_VEL
LIN {X 0,Y 64.896,Z 606.436,A -85,B 0,C 180,E1 -29200.706,E2 -29200.706} C_VEL
LIN {X 0,Y 56.682,Z 612.274,A -85,B 0,C 180,E1 -29211.688,E2 -29211.688} C_VEL
LIN {X 0,Y 50.894,Z 616.52,A -85,B 0,C 180,E1 -29225.527,E2 -29225.527} C_VEL
LIN {X 0,Y 48.388,Z 619.309,A -85,B 0,C 180,E1 -29241.649,E2 -29241.649} C_VEL
LIN {X 0,Y 48.363,Z 620.179,A -85,B 0,C 180,E1 -29250,E2 -29250} C_VEL
LIN {X 0,Y 49.276,Z 620.856,A -85,B 0,C 180,E1 -29266.574,E2 -29266.574} C_VEL
LIN {X 0,Y 53.506,Z 620.205,A -85,B 0,C 180,E1 -29281.696,E2 -29281.696} C_VEL
LIN {X 0,Y 60.783,Z 618.234,A -85,B 0,C 180,E1 -29293.928,E2 -29293.928} C_VEL
LIN {X 0,Y 70.093,Z 614.881,A -85,B 0,C 180,E1 -29303.335,E2 -29303.335} C_VEL
LIN {X 0,Y 80.923,Z 610.059,A -85,B 0,C 180,E1 -29310.283,E2 -29310.283} C_VEL
LIN {X 0,Y 92.639,Z 603.626,A -85,B 0,C 180,E1 -29315.559,E2 -29315.559} C_VEL
LIN {X 0,Y 103.48,Z 596.489,A -85,B 0,C 180,E1 -29319.046,E2 -29319.046} C_VEL
LIN {X 0,Y 113.972,Z 588.211,A -85,B 0,C 180,E1 -29321.762,E2 -29321.762} C_VEL
LIN {X 0,Y 124.283,Z 578.476,A -85,B 0,C 180,E1 -29324.014,E2 -29324.014} C_VEL
LIN {X 0,Y 133.336,Z 568.322,A -85,B 0,C 180,E1 -29325.589,E2 -29325.589} C_VEL
LIN {X 0,Y 141.649,Z 557.174,A -85,B 0,C 180,E1 -29326.834,E2 -29326.834} C_VEL
LIN {X 0,Y 149.205,Z 544.868,A -85,B 0,C 180,E1 -29327.794,E2 -29327.794} C_VEL
LIN {X 0,Y 155.126,Z 533.043,A -85,B 0,C 180,E1 -29328.445,E2 -29328.445} C_VEL
LIN {X 0,Y 159.6,Z 521.848,A -85,B 0,C 180,E1 -29328.961,E2 -29328.961} C_VEL
LIN {X 0,Y 163.895,Z 507.759,A -85,B 0,C 180,E1 -29329.407,E2 -29329.407} C_VEL
LIN {X 0,Y 166.208,Z 496.745,A -85,B 0,C 180,E1 -29329.727,E2 -29329.727} C_VEL
LIN {X 0,Y 165.709,Z 494.551,A -85,B 0,C 180,E1 -29332.384,E2 -29332.384} C_VEL
LIN {X 0,Y 165.457,Z 493.127,A -85,B 0,C 180,E1 -29334.516,E2 -29334.516} C_VEL
LIN {X 0,Y 165.251,Z 492.702,A -85,B 0,C 180,E1 -29337.563,E2 -29337.563} C_VEL
LIN {X 0,Y 165.488,Z 493.168,A -85,B 0,C 180,E1 -29341.217,E2 -29341.217} C_VEL
LIN {X 0,Y 165.629,Z 494.408,A -85,B 0,C 180,E1 -29342.852,E2 -29342.852} C_VEL
LIN {X 0,Y 165.549,Z 495.782,A -85,B 0,C 180,E1 -29343.519,E2 -29343.519} C_VEL
LIN {X 0,Y 165.166,Z 498.502,A -85,B 0,C 180,E1 -29344.016,E2 -29344.016} C_VEL
LIN {X 0,Y 164.548,Z 501.676,A -85,B 0,C 180,E1 -29344.208,E2 -29344.208} C_VEL
LIN {X 0,Y 161.259,Z 513.48,A -85,B 0,C 180,E1 -29343.848,E2 -29343.848} C_VEL
LIN {X 0,Y 160.778,Z 514.94,A -85,B 0,C 180,E1 -29343.88,E2 -29343.88} C_VEL
LIN {X 0,Y 155.658,Z 528.763,A -85,B 0,C 180,E1 -29344.434,E2 -29344.434} C_VEL
LIN {X 0,Y 149.061,Z 542.332,A -85,B 0,C 180,E1 -29345.115,E2 -29345.115} C_VEL
LIN {X 0,Y 142.586,Z 553.103,A -85,B 0,C 180,E1 -29345.94,E2 -29345.94} C_VEL
LIN {X 0,Y 134.553,Z 564.202,A -85,B 0,C 180,E1 -29347.057,E2 -29347.057} C_VEL
LIN {X 0,Y 126.076,Z 573.98,A -85,B 0,C 180,E1 -29348.323,E2 -29348.323} C_VEL
LIN {X 0,Y 116.032,Z 583.734,A -85,B 0,C 180,E1 -29350.179,E2 -29350.179} C_VEL
LIN {X 0,Y 106.157,Z 591.804,A -85,B 0,C 180,E1 -29352.442,E2 -29352.442} C_VEL
LIN {X 0,Y 94.803,Z 599.513,A -85,B 0,C 180,E1 -29355.478,E2 -29355.478} C_VEL
LIN {X 0,Y 85.352,Z 604.866,A -85,B 0,C 180,E1 -29358.756,E2 -29358.756} C_VEL
LIN {X 0,Y 76.252,Z 609.241,A -85,B 0,C 180,E1 -29362.825,E2 -29362.825} C_VEL
LIN {X 0,Y 64.888,Z 613.63,A -85,B 0,C 180,E1 -29369.947,E2 -29369.947} C_VEL
LIN {X 0,Y 54.892,Z 616.548,A -85,B 0,C 180,E1 -29379.807,E2 -29379.807} C_VEL
LIN {X 0,Y 46.9,Z 618.093,A -85,B 0,C 180,E1 -29393.172,E2 -29393.172} C_VEL
LIN {X 0,Y 42.157,Z 618.301,A -85,B 0,C 180,E1 -29410.523,E2 -29410.523} C_VEL
LIN {X 0,Y 41.248,Z 617.911,A -85,B 0,C 180,E1 -29420.189,E2 -29420.189} C_VEL
LIN {X 0,Y 41.29,Z 617.194,A -85,B 0,C 180,E1 -29430,E2 -29430} C_VEL
LIN {X 0,Y 44.088,Z 614.775,A -85,B 0,C 180,E1 -29448.591,E2 -29448.591} C_VEL
LIN {X 0,Y 50.242,Z 610.977,A -85,B 0,C 180,E1 -29464.024,E2 -29464.024} C_VEL
LIN {X 0,Y 56.58,Z 607.098,A -85,B 0,C 180,E1 -29473.092,E2 -29473.092} C_VEL
LIN {X 0,Y 66.496,Z 600.538,A -85,B 0,C 180,E1 -29482.436,E2 -29482.436} C_VEL
LIN {X 0,Y 76.284,Z 593.223,A -85,B 0,C 180,E1 -29488.451,E2 -29488.451} C_VEL
LIN {X 0,Y 86.724,Z 584.121,A -85,B 0,C 180,E1 -29493.053,E2 -29493.053} C_VEL
LIN {X 0,Y 95.976,Z 574.612,A -85,B 0,C 180,E1 -29496.254,E2 -29496.254} C_VEL
LIN {X 0,Y 104.548,Z 564.099,A -85,B 0,C 180,E1 -29498.862,E2 -29498.862} C_VEL
LIN {X 0,Y 112.615,Z 552.44,A -85,B 0,C 180,E1 -29500.72,E2 -29500.72} C_VEL
LIN {X 0,Y 119.1,Z 541.057,A -85,B 0,C 180,E1 -29502.088,E2 -29502.088} C_VEL
LIN {X 0,Y 124.847,Z 528.713,A -85,B 0,C 180,E1 -29503.133,E2 -29503.133} C_VEL
LIN {X 0,Y 129.83,Z 514.868,A -85,B 0,C 180,E1 -29504,E2 -29504} C_VEL
LIN {X 0,Y 133.436,Z 500.805,A -85,B 0,C 180,E1 -29504.677,E2 -29504.677} C_VEL
LIN {X 0,Y 135.726,Z 486.788,A -85,B 0,C 180,E1 -29505.07,E2 -29505.07} C_VEL
LIN {X 0,Y 136.804,Z 477.13,A -85,B 0,C 180,E1 -29505.34,E2 -29505.34} C_VEL
LIN {X 0,Y 135.698,Z 473.571,A -85,B 0,C 180,E1 -29508.99,E2 -29508.99} C_VEL
LIN {X 0,Y 135.05,Z 471.512,A -85,B 0,C 180,E1 -29512.26,E2 -29512.26} C_VEL
LIN {X 0,Y 134.839,Z 470.066,A -85,B 0,C 180,E1 -29514.766,E2 -29514.766} C_VEL
LIN {X 0,Y 134.876,Z 469.868,A -85,B 0,C 180,E1 -29519.999,E2 -29519.999} C_VEL
LIN {X 0,Y 135.698,Z 473.362,A -85,B 0,C 180,E1 -29525.572,E2 -29525.572} C_VEL
LIN {X 0,Y 136.833,Z 477.267,A -85,B 0,C 180,E1 -29529.39,E2 -29529.39} C_VEL
LIN {X 0,Y 134.125,Z 498.044,A -85,B 0,C 180,E1 -29529.933,E2 -29529.933} C_VEL
LIN {X 0,Y 130.792,Z 512.439,A -85,B 0,C 180,E1 -29530.392,E2 -29530.392} C_VEL
LIN {X 0,Y 126.216,Z 526.254,A -85,B 0,C 180,E1 -29531.067,E2 -29531.067} C_VEL
LIN {X 0,Y 120.361,Z 539.68,A -85,B 0,C 180,E1 -29532.025,E2 -29532.025} C_VEL
LIN {X 0,Y 113.71,Z 551.792,A -85,B 0,C 180,E1 -29533.232,E2 -29533.232} C_VEL
LIN {X 0,Y 105.47,Z 564.013,A -85,B 0,C 180,E1 -29534.936,E2 -29534.936} C_VEL
LIN {X 0,Y 96.924,Z 574.745,A -85,B 0,C 180,E1 -29537.317,E2 -29537.317} C_VEL
LIN {X 0,Y 87.93,Z 584.183,A -85,B 0,C 180,E1 -29540.092,E2 -29540.092} C_VEL
LIN {X 0,Y 78.684,Z 592.516,A -85,B 0,C 180,E1 -29543.72,E2 -29543.72} C_VEL
LIN {X 0,Y 68.53,Z 600.496,A -85,B 0,C 180,E1 -29549.343,E2 -29549.343} C_VEL
LIN {X 0,Y 60.456,Z 606.091,A -85,B 0,C 180,E1 -29555.536,E2 -29555.536} C_VEL
LIN {X 0,Y 51.263,Z 611.964,A -85,B 0,C 180,E1 -29566.727,E2 -29566.727} C_VEL
LIN {X 0,Y 44.485,Z 616.239,A -85,B 0,C 180,E1 -29581.708,E2 -29581.708} C_VEL
LIN {X 0,Y 41.368,Z 619.059,A -85,B 0,C 180,E1 -29600.219,E2 -29600.219} C_VEL
LIN {X 0,Y 41.274,Z 619.944,A -85,B 0,C 180,E1 -29610,E2 -29610} C_VEL
LIN {X 0,Y 42.501,Z 620.647,A -85,B 0,C 180,E1 -29629.313,E2 -29629.313} C_VEL
LIN {X 0,Y 47.572,Z 620.025,A -85,B 0,C 180,E1 -29646.224,E2 -29646.224} C_VEL
LIN {X 0,Y 55.851,Z 618.087,A -85,B 0,C 180,E1 -29659.027,E2 -29659.027} C_VEL
LIN {X 0,Y 66.083,Z 614.77,A -85,B 0,C 180,E1 -29668.302,E2 -29668.302} C_VEL
LIN {X 0,Y 77.626,Z 609.98,A -85,B 0,C 180,E1 -29674.874,E2 -29674.874} C_VEL
LIN {X 0,Y 89.921,Z 603.58,A -85,B 0,C 180,E1 -29679.702,E2 -29679.702} C_VEL
LIN {X 0,Y 101.155,Z 596.48,A -85,B 0,C 180,E1 -29682.809,E2 -29682.809} C_VEL
LIN {X 0,Y 111.379,Z 588.711,A -85,B 0,C 180,E1 -29685.111,E2 -29685.111} C_VEL
LIN {X 0,Y 120.86,Z 580.18,A -85,B 0,C 180,E1 -29686.911,E2 -29686.911} C_VEL
LIN {X 0,Y 130.908,Z 569.432,A -85,B 0,C 180,E1 -29688.461,E2 -29688.461} C_VEL
LIN {X 0,Y 140.207,Z 557.391,A -85,B 0,C 180,E1 -29689.651,E2 -29689.651} C_VEL
LIN {X 0,Y 147.868,Z 545.212,A -85,B 0,C 180,E1 -29690.481,E2 -29690.481} C_VEL
LIN {X 0,Y 153.866,Z 533.509,A -85,B 0,C 180,E1 -29691.025,E2 -29691.025} C_VEL
LIN {X 0,Y 158.27,Z 522.76,A -85,B 0,C 180,E1 -29691.461,E2 -29691.461} C_VEL
LIN {X 0,Y 162.743,Z 508.667,A -85,B 0,C 180,E1 -29691.857,E2 -29691.857} C_VEL
LIN {X 0,Y 164.36,Z 501.91,A -85,B 0,C 180,E1 -29692.029,E2 -29692.029} C_VEL
LIN {X 0,Y 164.162,Z 500.17,A -85,B 0,C 180,E1 -29694.473,E2 -29694.473} C_VEL
LIN {X 0,Y 163.972,Z 499.676,A -85,B 0,C 180,E1 -29697.544,E2 -29697.544} C_VEL
LIN {X 0,Y 164.136,Z 500.196,A -85,B 0,C 180,E1 -29701.074,E2 -29701.074} C_VEL
LIN {X 0,Y 164.258,Z 501.925,A -85,B 0,C 180,E1 -29703.452,E2 -29703.452} C_VEL
LIN {X 0,Y 160.778,Z 514.94,A -85,B 0,C 180,E1 -29703.88,E2 -29703.88} C_VEL
LIN {X 0,Y 158.809,Z 520.605,A -85,B 0,C 180,E1 -29703.839,E2 -29703.839} C_VEL
LIN {X 0,Y 154.933,Z 529.633,A -85,B 0,C 180,E1 -29703.154,E2 -29703.154} C_VEL
LIN {X 0,Y 150.629,Z 538.295,A -85,B 0,C 180,E1 -29702.447,E2 -29702.447} C_VEL
LIN {X 0,Y 147.825,Z 543.378,A -85,B 0,C 180,E1 -29702.442,E2 -29702.442} C_VEL
LIN {X 0,Y 140.781,Z 554.706,A -85,B 0,C 180,E1 -29703.202,E2 -29703.202} C_VEL
LIN {X 0,Y 132.135,Z 566.173,A -85,B 0,C 180,E1 -29704.226,E2 -29704.226} C_VEL
LIN {X 0,Y 123.522,Z 575.654,A -85,B 0,C 180,E1 -29705.312,E2 -29705.312} C_VEL
LIN {X 0,Y 113.281,Z 585.163,A -85,B 0,C 180,E1 -29706.949,E2 -29706.949} C_VEL
LIN {X 0,Y 101.483,Z 594.197,A -85,B 0,C 180,E1 -29709.297,E2 -29709.297} C_VEL
LIN {X 0,Y 89.844,Z 601.457,A -85,B 0,C 180,E1 -29712.091,E2 -29712.091} C_VEL
LIN {X 0,Y 79.474,Z 606.811,A -85,B 0,C 180,E1 -29715.386,E2 -29715.386} C_VEL
LIN {X 0,Y 67.576,Z 611.735,A -85,B 0,C 180,E1 -29720.605,E2 -29720.605} C_VEL
LIN {X 0,Y 55.933,Z 615.405,A -85,B 0,C 180,E1 -29728.41,E2 -29728.41} C_VEL
LIN {X 0,Y 45.681,Z 617.657,A -85,B 0,C 180,E1 -29739.713,E2 -29739.713} C_VEL
LIN {X 0,Y 37.877,Z 618.561,A -85,B 0,C 180,E1 -29756.176,E2 -29756.176} C_VEL
LIN {X 0,Y 34.224,Z 618.135,A -85,B 0,C 180,E1 -29778.149,E2 -29778.149} C_VEL
LIN {X 0,Y 34.163,Z 617.432,A -85,B 0,C 180,E1 -29790,E2 -29790} C_VEL
LIN {X 0,Y 37.453,Z 615.04,A -85,B 0,C 180,E1 -29812.042,E2 -29812.042} C_VEL
LIN {X 0,Y 44.556,Z 611.274,A -85,B 0,C 180,E1 -29829.119,E2 -29829.119} C_VEL
LIN {X 0,Y 51.634,Z 607.425,A -85,B 0,C 180,E1 -29838.47,E2 -29838.47} C_VEL
LIN {X 0,Y 62.438,Z 600.897,A -85,B 0,C 180,E1 -29847.586,E2 -29847.586} C_VEL
LIN {X 0,Y 72.835,Z 593.625,A -85,B 0,C 180,E1 -29853.195,E2 -29853.195} C_VEL
LIN {X 0,Y 83.757,Z 584.583,A -85,B 0,C 180,E1 -29857.37,E2 -29857.37} C_VEL
LIN {X 0,Y 93.35,Z 575.126,A -85,B 0,C 180,E1 -29860.235,E2 -29860.235} C_VEL
LIN {X 0,Y 102.212,Z 564.676,A -85,B 0,C 180,E1 -29862.561,E2 -29862.561} C_VEL
LIN {X 0,Y 110.483,Z 553.095,A -85,B 0,C 180,E1 -29864.182,E2 -29864.182} C_VEL
LIN {X 0,Y 117.964,Z 540.238,A -85,B 0,C 180,E1 -29865.498,E2 -29865.498} C_VEL
LIN {X 0,Y 123.75,Z 527.81,A -85,B 0,C 180,E1 -29866.394,E2 -29866.394} C_VEL
LIN {X 0,Y 128.54,Z 514.514,A -85,B 0,C 180,E1 -29867.109,E2 -29867.109} C_VEL
LIN {X 0,Y 132.141,Z 500.584,A -85,B 0,C 180,E1 -29867.694,E2 -29867.694} C_VEL
LIN {X 0,Y 134.536,Z 485.642,A -85,B 0,C 180,E1 -29868.057,E2 -29868.057} C_VEL
LIN {X 0,Y 134.968,Z 481.639,A -85,B 0,C 180,E1 -29868.233,E2 -29868.233} C_VEL
LIN {X 0,Y 134.306,Z 479.248,A -85,B 0,C 180,E1 -29871.325,E2 -29871.325} C_VEL
LIN {X 0,Y 133.956,Z 477.18,A -85,B 0,C 180,E1 -29874.845,E2 -29874.845} C_VEL
LIN {X 0,Y 133.874,Z 476.86,A -85,B 0,C 180,E1 -29876.99,E2 -29876.99} C_VEL
LIN {X 0,Y 134.005,Z 477.167,A -85,B 0,C 180,E1 -29880.234,E2 -29880.234} C_VEL
LIN {X 0,Y 134.615,Z 480.235,A -85,B 0,C 180,E1 -29884.866,E2 -29884.866} C_VEL
LIN {X 0,Y 135.005,Z 481.815,A -85,B 0,C 180,E1 -29886.561,E2 -29886.561} C_VEL
LIN {X 0,Y 132.484,Z 499.463,A -85,B 0,C 180,E1 -29886.984,E2 -29886.984} C_VEL
LIN {X 0,Y 129.174,Z 513.048,A -85,B 0,C 180,E1 -29887.355,E2 -29887.355} C_VEL
LIN {X 0,Y 124.617,Z 526.406,A -85,B 0,C 180,E1 -29887.916,E2 -29887.916} C_VEL
LIN {X 0,Y 119.082,Z 538.871,A -85,B 0,C 180,E1 -29888.676,E2 -29888.676} C_VEL
LIN {X 0,Y 112.292,Z 551.11,A -85,B 0,C 180,E1 -29889.686,E2 -29889.686} C_VEL
LIN {X 0,Y 103.852,Z 563.437,A -85,B 0,C 180,E1 -29891.108,E2 -29891.108} C_VEL
LIN {X 0,Y 95.395,Z 573.852,A -85,B 0,C 180,E1 -29893.121,E2 -29893.121} C_VEL
LIN {X 0,Y 85.738,Z 583.722,A -85,B 0,C 180,E1 -29895.601,E2 -29895.601} C_VEL
LIN {X 0,Y 76.083,Z 592.098,A -85,B 0,C 180,E1 -29898.77,E2 -29898.77} C_VEL
LIN {X 0,Y 65.317,Z 600.118,A -85,B 0,C 180,E1 -29903.853,E2 -29903.853} C_VEL
LIN {X 0,Y 55.942,Z 606.134,A -85,B 0,C 180,E1 -29910.165,E2 -29910.165} C_VEL
LIN {X 0,Y 46.304,Z 611.652,A -85,B 0,C 180,E1 -29920.633,E2 -29920.633} C_VEL
LIN {X 0,Y 38.327,Z 615.959,A -85,B 0,C 180,E1 -29936.626,E2 -29936.626} C_VEL
LIN {X 0,Y 34.366,Z 618.808,A -85,B 0,C 180,E1 -29958.2,E2 -29958.2} C_VEL
LIN {X 0,Y 34.159,Z 619.707,A -85,B 0,C 180,E1 -29970,E2 -29970} C_VEL
LIN {X 0,Y 35.839,Z 620.437,A -85,B 0,C 180,E1 -29993.092,E2 -29993.092} C_VEL
LIN {X 0,Y 42.021,Z 619.843,A -85,B 0,C 180,E1 -30011.99,E2 -30011.99} C_VEL
LIN {X 0,Y 51.446,Z 617.936,A -85,B 0,C 180,E1 -30025.052,E2 -30025.052} C_VEL
LIN {X 0,Y 62.622,Z 614.658,A -85,B 0,C 180,E1 -30033.875,E2 -30033.875} C_VEL
LIN {X 0,Y 74.876,Z 609.9,A -85,B 0,C 180,E1 -30039.822,E2 -30039.822} C_VEL
LIN {X 0,Y 87.704,Z 603.534,A -85,B 0,C 180,E1 -30044.072,E2 -30044.072} C_VEL
LIN {X 0,Y 99.286,Z 596.471,A -85,B 0,C 180,E1 -30046.732,E2 -30046.732} C_VEL
LIN {X 0,Y 109.479,Z 588.975,A -85,B 0,C 180,E1 -30048.652,E2 -30048.652} C_VEL
LIN {X 0,Y 119.45,Z 580.259,A -85,B 0,C 180,E1 -30050.238,E2 -30050.238} C_VEL
LIN {X 0,Y 129.677,Z 569.567,A -85,B 0,C 180,E1 -30051.529,E2 -30051.529} C_VEL
LIN {X 0,Y 138.25,Z 558.765,A -85,B 0,C 180,E1 -30052.436,E2 -30052.436} C_VEL
LIN {X 0,Y 146.004,Z 546.961,A -85,B 0,C 180,E1 -30053.124,E2 -30053.124} C_VEL
LIN {X 0,Y 152.923,Z 533.93,A -85,B 0,C 180,E1 -30053.641,E2 -30053.641} C_VEL
LIN {X 0,Y 157.821,Z 522.179,A -85,B 0,C 180,E1 -30054.038,E2 -30054.038} C_VEL
LIN {X 0,Y 162.28,Z 508.16,A -85,B 0,C 180,E1 -30054.355,E2 -30054.355} C_VEL
LIN {X 0,Y 162.483,Z 507.32,A -85,B 0,C 180,E1 -30054.477,E2 -30054.477} C_VEL
LIN {X 0,Y 162.484,Z 506.95,A -85,B 0,C 180,E1 -30055.038,E2 -30055.038} C_VEL
LIN {X 0,Y 162.362,Z 506.67,A -85,B 0,C 180,E1 -30058.761,E2 -30058.761} C_VEL
LIN {X 0,Y 162.433,Z 507.234,A -85,B 0,C 180,E1 -30060.961,E2 -30060.961} C_VEL
LIN {X 0,Y 162.341,Z 507.661,A -85,B 0,C 180,E1 -30061.129,E2 -30061.129} C_VEL
LIN {X 0,Y 157.738,Z 522.071,A -85,B 0,C 180,E1 -30061.589,E2 -30061.589} C_VEL
LIN {X 0,Y 152.082,Z 535.243,A -85,B 0,C 180,E1 -30062.075,E2 -30062.075} C_VEL
LIN {X 0,Y 147.825,Z 543.378,A -85,B 0,C 180,E1 -30062.442,E2 -30062.442} C_VEL
LIN {X 0,Y 144.835,Z 548.482,A -85,B 0,C 180,E1 -30062.476,E2 -30062.476} C_VEL
LIN {X 0,Y 139.318,Z 556.593,A -85,B 0,C 180,E1 -30061.874,E2 -30061.874} C_VEL
LIN {X 0,Y 133.264,Z 564.298,A -85,B 0,C 180,E1 -30061.267,E2 -30061.267} C_VEL
LIN {X 0,Y 129.407,Z 568.763,A -85,B 0,C 180,E1 -30061.349,E2 -30061.349} C_VEL
LIN {X 0,Y 119.581,Z 578.919,A -85,B 0,C 180,E1 -30062.39,E2 -30062.39} C_VEL
LIN {X 0,Y 108.801,Z 588.176,A -85,B 0,C 180,E1 -30063.872,E2 -30063.872} C_VEL
LIN {X 0,Y 97.141,Z 596.436,A -85,B 0,C 180,E1 -30065.845,E2 -30065.845} C_VEL
LIN {X 0,Y 85.234,Z 603.307,A -85,B 0,C 180,E1 -30068.32,E2 -30068.32} C_VEL
LIN {X 0,Y 74.426,Z 608.362,A -85,B 0,C 180,E1 -30071.322,E2 -30071.322} C_VEL
LIN {X 0,Y 62.184,Z 612.903,A -85,B 0,C 180,E1 -30076.12,E2 -30076.12} C_VEL
LIN {X 0,Y 52.885,Z 615.544,A -85,B 0,C 180,E1 -30081.525,E2 -30081.525} C_VEL
LIN {X 0,Y 41.464,Z 617.826,A -85,B 0,C 180,E1 -30092.059,E2 -30092.059} C_VEL
LIN {X 0,Y 32.161,Z 618.757,A -85,B 0,C 180,E1 -30109.035,E2 -30109.035} C_VEL
LIN {X 0,Y 27.276,Z 618.359,A -85,B 0,C 180,E1 -30135.068,E2 -30135.068} C_VEL
LIN {X 0,Y 27.042,Z 617.669,A -85,B 0,C 180,E1 -30149.999,E2 -30149.999} C_VEL
LIN {X 0,Y 30.988,Z 615.305,A -85,B 0,C 180,E1 -30176.974,E2 -30176.974} C_VEL
LIN {X 0,Y 39.315,Z 611.568,A -85,B 0,C 180,E1 -30195.647,E2 -30195.647} C_VEL
LIN {X 0,Y 47.242,Z 607.75,A -85,B 0,C 180,E1 -30204.906,E2 -30204.906} C_VEL
LIN {X 0,Y 58.941,Z 601.258,A -85,B 0,C 180,E1 -30213.416,E2 -30213.416} C_VEL
LIN {X 0,Y 69.926,Z 594.023,A -85,B 0,C 180,E1 -30218.386,E2 -30218.386} C_VEL
LIN {X 0,Y 81.298,Z 585.045,A -85,B 0,C 180,E1 -30221.975,E2 -30221.975} C_VEL
LIN {X 0,Y 91.202,Z 575.64,A -85,B 0,C 180,E1 -30224.419,E2 -30224.419} C_VEL
LIN {X 0,Y 100.319,Z 565.253,A -85,B 0,C 180,E1 -30226.419,E2 -30226.419} C_VEL
LIN {X 0,Y 108.769,Z 553.75,A -85,B 0,C 180,E1 -30227.765,E2 -30227.765} C_VEL
LIN {X 0,Y 116.399,Z 540.993,A -85,B 0,C 180,E1 -30228.86,E2 -30228.86} C_VEL
LIN {X 0,Y 122.255,Z 528.776,A -85,B 0,C 180,E1 -30229.601,E2 -30229.601} C_VEL
LIN {X 0,Y 127.214,Z 515.443,A -85,B 0,C 180,E1 -30230.214,E2 -30230.214} C_VEL
LIN {X 0,Y 130.87,Z 501.853,A -85,B 0,C 180,E1 -30230.722,E2 -30230.722} C_VEL
LIN {X 0,Y 133.286,Z 487.985,A -85,B 0,C 180,E1 -30231.017,E2 -30231.017} C_VEL
LIN {X 0,Y 133.443,Z 486.687,A -85,B 0,C 180,E1 -30231.099,E2 -30231.099} C_VEL
LIN {X 0,Y 133.039,Z 484.074,A -85,B 0,C 180,E1 -30235.684,E2 -30235.684} C_VEL
LIN {X 0,Y 133.092,Z 484.196,A -85,B 0,C 180,E1 -30239.794,E2 -30239.794} C_VEL
LIN {X 0,Y 133.47,Z 486.59,A -85,B 0,C 180,E1 -30243.6,E2 -30243.6} C_VEL
LIN {X 0,Y 131.12,Z 501.265,A -85,B 0,C 180,E1 -30243.966,E2 -30243.966} C_VEL
LIN {X 0,Y 127.476,Z 515.133,A -85,B 0,C 180,E1 -30244.301,E2 -30244.301} C_VEL
LIN {X 0,Y 122.536,Z 528.632,A -85,B 0,C 180,E1 -30244.769,E2 -30244.769} C_VEL
LIN {X 0,Y 116.486,Z 541.393,A -85,B 0,C 180,E1 -30245.434,E2 -30245.434} C_VEL
LIN {X 0,Y 108.73,Z 554.399,A -85,B 0,C 180,E1 -30246.383,E2 -30246.383} C_VEL
LIN {X 0,Y 101.007,Z 565.02,A -85,B 0,C 180,E1 -30247.47,E2 -30247.47} C_VEL
LIN {X 0,Y 92.542,Z 574.913,A -85,B 0,C 180,E1 -30249.149,E2 -30249.149} C_VEL
LIN {X 0,Y 82.421,Z 584.76,A -85,B 0,C 180,E1 -30251.302,E2 -30251.302} C_VEL
LIN {X 0,Y 72.444,Z 592.924,A -85,B 0,C 180,E1 -30254.038,E2 -30254.038} C_VEL
LIN {X 0,Y 61.181,Z 600.759,A -85,B 0,C 180,E1 -30258.612,E2 -30258.612} C_VEL
LIN {X 0,Y 50.623,Z 606.929,A -85,B 0,C 180,E1 -30264.898,E2 -30264.898} C_VEL
LIN {X 0,Y 41.983,Z 611.341,A -85,B 0,C 180,E1 -30273.174,E2 -30273.174} C_VEL
LIN {X 0,Y 32.587,Z 615.678,A -85,B 0,C 180,E1 -30289.683,E2 -30289.683} C_VEL
LIN {X 0,Y 27.418,Z 618.557,A -85,B 0,C 180,E1 -30315.148,E2 -30315.148} C_VEL
LIN {X 0,Y 27.048,Z 619.471,A -85,B 0,C 180,E1 -30330.001,E2 -30330.001} C_VEL
LIN {X 0,Y 29.412,Z 620.227,A -85,B 0,C 180,E1 -30358.549,E2 -30358.549} C_VEL
LIN {X 0,Y 37.026,Z 619.661,A -85,B 0,C 180,E1 -30379.4,E2 -30379.4} C_VEL
LIN {X 0,Y 47.712,Z 617.782,A -85,B 0,C 180,E1 -30392.106,E2 -30392.106} C_VEL
LIN {X 0,Y 59.825,Z 614.542,A -85,B 0,C 180,E1 -30400.022,E2 -30400.022} C_VEL
LIN {X 0,Y 72.727,Z 609.821,A -85,B 0,C 180,E1 -30405.098,E2 -30405.098} C_VEL
LIN {X 0,Y 86.024,Z 603.488,A -85,B 0,C 180,E1 -30408.635,E2 -30408.635} C_VEL
LIN {X 0,Y 97.896,Z 596.461,A -85,B 0,C 180,E1 -30410.798,E2 -30410.798} C_VEL
LIN {X 0,Y 109.446,Z 588.107,A -85,B 0,C 180,E1 -30412.484,E2 -30412.484} C_VEL
LIN {X 0,Y 120.172,Z 578.712,A -85,B 0,C 180,E1 -30413.835,E2 -30413.835} C_VEL
LIN {X 0,Y 130.556,Z 567.752,A -85,B 0,C 180,E1 -30414.803,E2 -30414.803} C_VEL
LIN {X 0,Y 139.233,Z 556.614,A -85,B 0,C 180,E1 -30415.503,E2 -30415.503} C_VEL
LIN {X 0,Y 147.069,Z 544.319,A -85,B 0,C 180,E1 -30415.997,E2 -30415.997} C_VEL
LIN {X 0,Y 153.172,Z 532.51,A -85,B 0,C 180,E1 -30416.347,E2 -30416.347} C_VEL
LIN {X 0,Y 157.723,Z 521.517,A -85,B 0,C 180,E1 -30416.621,E2 -30416.621} C_VEL
LIN {X 0,Y 159.822,Z 515.435,A -85,B 0,C 180,E1 -30416.736,E2 -30416.736} C_VEL
LIN {X 0,Y 160.429,Z 513.498,A -85,B 0,C 180,E1 -30417.111,E2 -30417.111} C_VEL
LIN {X 0,Y 160.426,Z 513.484,A -85,B 0,C 180,E1 -30418.686,E2 -30418.686} C_VEL
LIN {X 0,Y 156.508,Z 524.55,A -85,B 0,C 180,E1 -30419.089,E2 -30419.089} C_VEL
LIN {X 0,Y 151.11,Z 536.595,A -85,B 0,C 180,E1 -30419.448,E2 -30419.448} C_VEL
LIN {X 0,Y 144.733,Z 548.031,A -85,B 0,C 180,E1 -30419.899,E2 -30419.899} C_VEL
LIN {X 0,Y 137.055,Z 559.336,A -85,B 0,C 180,E1 -30420.607,E2 -30420.607} C_VEL
LIN {X 0,Y 129.407,Z 568.763,A -85,B 0,C 180,E1 -30421.349,E2 -30421.349} C_VEL
LIN {X 0,Y 125.37,Z 573.153,A -85,B 0,C 180,E1 -30421.44,E2 -30421.44} C_VEL
LIN {X 0,Y 118.289,Z 579.99,A -85,B 0,C 180,E1 -30420.787,E2 -30420.787} C_VEL
LIN {X 0,Y 110.851,Z 586.366,A -85,B 0,C 180,E1 -30420.153,E2 -30420.153} C_VEL
LIN {X 0,Y 106.239,Z 589.904,A -85,B 0,C 180,E1 -30420.37,E2 -30420.37} C_VEL
LIN {X 0,Y 94.928,Z 597.555,A -85,B 0,C 180,E1 -30421.851,E2 -30421.851} C_VEL
LIN {X 0,Y 84.493,Z 603.35,A -85,B 0,C 180,E1 -30423.481,E2 -30423.481} C_VEL
LIN {X 0,Y 75.073,Z 607.726,A -85,B 0,C 180,E1 -30425.373,E2 -30425.373} C_VEL
LIN {X 0,Y 63.945,Z 611.954,A -85,B 0,C 180,E1 -30428.439,E2 -30428.439} C_VEL
LIN {X 0,Y 50.686,Z 615.684,A -85,B 0,C 180,E1 -30433.923,E2 -30433.923} C_VEL
LIN {X 0,Y 38.143,Z 617.993,A -85,B 0,C 180,E1 -30442.886,E2 -30442.886} C_VEL
LIN {X 0,Y 27.153,Z 618.954,A -85,B 0,C 180,E1 -30459.057,E2 -30459.057} C_VEL
LIN {X 0,Y 20.44,Z 618.583,A -85,B 0,C 180,E1 -30489.888,E2 -30489.888} C_VEL
LIN {X 0,Y 19.936,Z 617.906,A -85,B 0,C 180,E1 -30509.999,E2 -30509.999} C_VEL
LIN {X 0,Y 24.883,Z 615.57,A -85,B 0,C 180,E1 -30544.394,E2 -30544.394} C_VEL
LIN {X 0,Y 34.728,Z 611.863,A -85,B 0,C 180,E1 -30564.045,E2 -30564.045} C_VEL
LIN {X 0,Y 43.558,Z 608.077,A -85,B 0,C 180,E1 -30572.55,E2 -30572.55} C_VEL
LIN {X 0,Y 56.131,Z 601.618,A -85,B 0,C 180,E1 -30579.894,E2 -30579.894} C_VEL
LIN {X 0,Y 67.635,Z 594.421,A -85,B 0,C 180,E1 -30583.982,E2 -30583.982} C_VEL
LIN {X 0,Y 79.396,Z 585.506,A -85,B 0,C 180,E1 -30586.832,E2 -30586.832} C_VEL
LIN {X 0,Y 89.562,Z 576.154,A -85,B 0,C 180,E1 -30588.78,E2 -30588.78} C_VEL
LIN {X 0,Y 98.901,Z 565.828,A -85,B 0,C 180,E1 -30590.394,E2 -30590.394} C_VEL
LIN {X 0,Y 107.494,Z 554.405,A -85,B 0,C 180,E1 -30591.448,E2 -30591.448} C_VEL
LIN {X 0,Y 115.242,Z 541.75,A -85,B 0,C 180,E1 -30592.309,E2 -30592.309} C_VEL
LIN {X 0,Y 121.148,Z 529.751,A -85,B 0,C 180,E1 -30592.876,E2 -30592.876} C_VEL
LIN {X 0,Y 126.21,Z 516.554,A -85,B 0,C 180,E1 -30593.36,E2 -30593.36} C_VEL
LIN {X 0,Y 130.06,Z 502.755,A -85,B 0,C 180,E1 -30593.795,E2 -30593.795} C_VEL
LIN {X 0,Y 132.085,Z 492.192,A -85,B 0,C 180,E1 -30594.082,E2 -30594.082} C_VEL
LIN {X 0,Y 132.072,Z 491.057,A -85,B 0,C 180,E1 -30596.185,E2 -30596.185} C_VEL
LIN {X 0,Y 132.108,Z 491.16,A -85,B 0,C 180,E1 -30599.237,E2 -30599.237} C_VEL
LIN {X 0,Y 132.136,Z 492.003,A -85,B 0,C 180,E1 -30600.661,E2 -30600.661} C_VEL
LIN {X 0,Y 129.3,Z 506.209,A -85,B 0,C 180,E1 -30600.962,E2 -30600.962} C_VEL
LIN {X 0,Y 125.215,Z 519.775,A -85,B 0,C 180,E1 -30601.226,E2 -30601.226} C_VEL
LIN {X 0,Y 119.526,Z 533.687,A -85,B 0,C 180,E1 -30601.651,E2 -30601.651} C_VEL
LIN {X 0,Y 112.533,Z 546.843,A -85,B 0,C 180,E1 -30602.222,E2 -30602.222} C_VEL
LIN {X 0,Y 104.68,Z 558.749,A -85,B 0,C 180,E1 -30602.947,E2 -30602.947} C_VEL
LIN {X 0,Y 97.056,Z 568.44,A -85,B 0,C 180,E1 -30603.904,E2 -30603.904} C_VEL
LIN {X 0,Y 88.217,Z 577.946,A -85,B 0,C 180,E1 -30605.228,E2 -30605.228} C_VEL
LIN {X 0,Y 77.887,Z 587.226,A -85,B 0,C 180,E1 -30606.989,E2 -30606.989} C_VEL
LIN {X 0,Y 67.665,Z 594.962,A -85,B 0,C 180,E1 -30609.348,E2 -30609.348} C_VEL
LIN {X 0,Y 57.626,Z 601.4,A -85,B 0,C 180,E1 -30612.665,E2 -30612.665} C_VEL
LIN {X 0,Y 48.651,Z 606.279,A -85,B 0,C 180,E1 -30616.791,E2 -30616.791} C_VEL
LIN {X 0,Y 38.527,Z 611.029,A -85,B 0,C 180,E1 -30624.206,E2 -30624.206} C_VEL
LIN {X 0,Y 27.522,Z 615.397,A -85,B 0,C 180,E1 -30639.997,E2 -30639.997} C_VEL
LIN {X 0,Y 20.613,Z 618.306,A -85,B 0,C 180,E1 -30670.066,E2 -30670.066} C_VEL
LIN {X 0,Y 19.951,Z 619.235,A -85,B 0,C 180,E1 -30690.001,E2 -30690.001} C_VEL
LIN {X 0,Y 23.403,Z 620.018,A -85,B 0,C 180,E1 -30726.914,E2 -30726.914} C_VEL
LIN {X 0,Y 32.834,Z 619.479,A -85,B 0,C 180,E1 -30748.892,E2 -30748.892} C_VEL
LIN {X 0,Y 44.816,Z 617.628,A -85,B 0,C 180,E1 -30760.207,E2 -30760.207} C_VEL
LIN {X 0,Y 57.778,Z 614.422,A -85,B 0,C 180,E1 -30766.685,E2 -30766.685} C_VEL
LIN {X 0,Y 71.226,Z 609.742,A -85,B 0,C 180,E1 -30770.655,E2 -30770.655} C_VEL
LIN {X 0,Y 84.909,Z 603.443,A -85,B 0,C 180,E1 -30773.344,E2 -30773.344} C_VEL
LIN {X 0,Y 97.012,Z 596.452,A -85,B 0,C 180,E1 -30774.956,E2 -30774.956} C_VEL
LIN {X 0,Y 108.02,Z 588.703,A -85,B 0,C 180,E1 -30776.131,E2 -30776.131} C_VEL
LIN {X 0,Y 119.619,Z 578.791,A -85,B 0,C 180,E1 -30777.214,E2 -30777.214} C_VEL
LIN {X 0,Y 126.608,Z 571.785,A -85,B 0,C 180,E1 -30777.692,E2 -30777.692} C_VEL
LIN {X 0,Y 126.556,Z 571.814,A -85,B 0,C 180,E1 -30778.381,E2 -30778.381} C_VEL
LIN {X 0,Y 115.972,Z 582.06,A -85,B 0,C 180,E1 -30779.28,E2 -30779.28} C_VEL
LIN {X 0,Y 106.239,Z 589.904,A -85,B 0,C 180,E1 -30780.37,E2 -30780.37} C_VEL
LIN {X 0,Y 100.751,Z 593.845,A -85,B 0,C 180,E1 -30780.725,E2 -30780.725} C_VEL
LIN {X 0,Y 91.12,Z 599.848,A -85,B 0,C 180,E1 -30780.224,E2 -30780.224} C_VEL
LIN {X 0,Y 83.086,Z 604.086,A -85,B 0,C 180,E1 -30779.611,E2 -30779.611} C_VEL
LIN {X 0,Y 76.894,Z 606.911,A -85,B 0,C 180,E1 -30779.648,E2 -30779.648} C_VEL
LIN {X 0,Y 74.815,Z 607.774,A -85,B 0,C 180,E1 -30779.864,E2 -30779.864} C_VEL
LIN {X 0,Y 63.29,Z 612.063,A -85,B 0,C 180,E1 -30781.955,E2 -30781.955} C_VEL
LIN {X 0,Y 49.447,Z 615.824,A -85,B 0,C 180,E1 -30785.774,E2 -30785.774} C_VEL
LIN {X 0,Y 35.96,Z 618.162,A -85,B 0,C 180,E1 -30792.258,E2 -30792.258} C_VEL
LIN {X 0,Y 23.31,Z 619.15,A -85,B 0,C 180,E1 -30805.241,E2 -30805.241} C_VEL
LIN {X 0,Y 13.947,Z 618.808,A -85,B 0,C 180,E1 -30839.739,E2 -30839.739} C_VEL
LIN {X 0,Y 12.817,Z 618.144,A -85,B 0,C 180,E1 -30869.999,E2 -30869.999} C_VEL
LIN {X 0,Y 19.449,Z 615.835,A -85,B 0,C 180,E1 -30916.279,E2 -30916.279} C_VEL
LIN {X 0,Y 31.105,Z 612.158,A -85,B 0,C 180,E1 -30934.659,E2 -30934.659} C_VEL
LIN {X 0,Y 40.778,Z 608.403,A -85,B 0,C 180,E1 -30941.425,E2 -30941.425} C_VEL
LIN {X 0,Y 54.108,Z 601.978,A -85,B 0,C 180,E1 -30946.949,E2 -30946.949} C_VEL
LIN {X 0,Y 66.031,Z 594.819,A -85,B 0,C 180,E1 -30949.908,E2 -30949.908} C_VEL
LIN {X 0,Y 78.09,Z 585.959,A -85,B 0,C 180,E1 -30951.886,E2 -30951.886} C_VEL
LIN {X 0,Y 88.459,Z 576.667,A -85,B 0,C 180,E1 -30953.276,E2 -30953.276} C_VEL
LIN {X 0,Y 98.834,Z 565.346,A -85,B 0,C 180,E1 -30954.581,E2 -30954.581} C_VEL
LIN {X 0,Y 107.541,Z 553.778,A -85,B 0,C 180,E1 -30955.286,E2 -30955.286} C_VEL
LIN {X 0,Y 115.385,Z 540.931,A -85,B 0,C 180,E1 -30955.861,E2 -30955.861} C_VEL
LIN {X 0,Y 121.803,Z 527.644,A -85,B 0,C 180,E1 -30956.297,E2 -30956.297} C_VEL
LIN {X 0,Y 126.72,Z 514.315,A -85,B 0,C 180,E1 -30956.657,E2 -30956.657} C_VEL
LIN {X 0,Y 130.396,Z 500.377,A -85,B 0,C 180,E1 -30956.956,E2 -30956.956} C_VEL
LIN {X 0,Y 130.863,Z 497.951,A -85,B 0,C 180,E1 -30957.043,E2 -30957.043} C_VEL
LIN {X 0,Y 130.867,Z 497.947,A -85,B 0,C 180,E1 -30957.67,E2 -30957.67} C_VEL
LIN {X 0,Y 127.527,Z 511.616,A -85,B 0,C 180,E1 -30957.87,E2 -30957.87} C_VEL
LIN {X 0,Y 122.691,Z 525.538,A -85,B 0,C 180,E1 -30958.082,E2 -30958.082} C_VEL
LIN {X 0,Y 116.887,Z 538.207,A -85,B 0,C 180,E1 -30958.389,E2 -30958.389} C_VEL
LIN {X 0,Y 109.84,Z 550.451,A -85,B 0,C 180,E1 -30958.733,E2 -30958.733} C_VEL
LIN {X 0,Y 101.037,Z 562.791,A -85,B 0,C 180,E1 -30959.251,E2 -30959.251} C_VEL
LIN {X 0,Y 91.365,Z 573.887,A -85,B 0,C 180,E1 -30960.243,E2 -30960.243} C_VEL
LIN {X 0,Y 80.844,Z 583.839,A -85,B 0,C 180,E1 -30961.319,E2 -30961.319} C_VEL
LIN {X 0,Y 70.355,Z 592.09,A -85,B 0,C 180,E1 -30962.65,E2 -30962.65} C_VEL
LIN {X 0,Y 58.214,Z 600.002,A -85,B 0,C 180,E1 -30965.127,E2 -30965.127} C_VEL
LIN {X 0,Y 46.183,Z 606.368,A -85,B 0,C 180,E1 -30968.751,E2 -30968.751} C_VEL
LIN {X 0,Y 32.926,Z 611.976,A -85,B 0,C 180,E1 -30976.155,E2 -30976.155} C_VEL
LIN {X 0,Y 23.57,Z 615.117,A -85,B 0,C 180,E1 -30986.551,E2 -30986.551} C_VEL
LIN {X 0,Y 14.134,Z 618.056,A -85,B 0,C 180,E1 -31020.184,E2 -31020.184} C_VEL
LIN {X 0,Y 12.842,Z 618.998,A -85,B 0,C 180,E1 -31050.001,E2 -31050.001} C_VEL
LIN {X 0,Y 18.21,Z 619.809,A -85,B 0,C 180,E1 -31100.527,E2 -31100.527} C_VEL
LIN {X 0,Y 29.784,Z 619.297,A -85,B 0,C 180,E1 -31120.715,E2 -31120.715} C_VEL
LIN {X 0,Y 42.927,Z 617.474,A -85,B 0,C 180,E1 -31129.214,E2 -31129.214} C_VEL
LIN {X 0,Y 56.562,Z 614.298,A -85,B 0,C 180,E1 -31133.739,E2 -31133.739} C_VEL
LIN {X 0,Y 70.419,Z 609.662,A -85,B 0,C 180,E1 -31136.406,E2 -31136.406} C_VEL
LIN {X 0,Y 80.883,Z 605.12,A -85,B 0,C 180,E1 -31137.781,E2 -31137.781} C_VEL
LIN {X 0,Y 84.381,Z 603.397,A -85,B 0,C 180,E1 -31138.14,E2 -31138.14} C_VEL
LIN {X 0,Y 84.362,Z 603.392,A -85,B 0,C 180,E1 -31138.608,E2 -31138.608} C_VEL
LIN {X 0,Y 74.815,Z 607.774,A -85,B 0,C 180,E1 -31139.864,E2 -31139.864} C_VEL
LIN {X 0,Y 69.097,Z 610.037,A -85,B 0,C 180,E1 -31140.485,E2 -31140.485} C_VEL
LIN {X 0,Y 57.352,Z 613.876,A -85,B 0,C 180,E1 -31140.95,E2 -31140.95} C_VEL
LIN {X 0,Y 45.33,Z 616.753,A -85,B 0,C 180,E1 -31140.932,E2 -31140.932} C_VEL
LIN {X 0,Y 39.243,Z 617.82,A -85,B 0,C 180,E1 -31141.117,E2 -31141.117} C_VEL
LIN {X 0,Y 33.143,Z 618.596,A -85,B 0,C 180,E1 -31141.856,E2 -31141.856} C_VEL
LIN {X 0,Y 27.084,Z 619.058,A -85,B 0,C 180,E1 -31143.822,E2 -31143.822} C_VEL
LIN {X 0,Y 14.579,Z 619.355,A -85,B 0,C 180,E1 -31155.388,E2 -31155.388} C_VEL
LIN {X 0,Y 5.69,Z 618.382,A -85,B 0,C 180,E1 -31229.997,E2 -31229.997} C_VEL
LIN {X 0,Y 9.335,Z 617.407,A -85,B 0,C 180,E1 -31278.836,E2 -31278.836} C_VEL
LIN {X 0,Y 15.421,Z 616.101,A -85,B 0,C 180,E1 -31295.713,E2 -31295.713} C_VEL
LIN {X 0,Y 28.798,Z 612.452,A -85,B 0,C 180,E1 -31307.47,E2 -31307.47} C_VEL
LIN {X 0,Y 42.556,Z 607.319,A -85,B 0,C 180,E1 -31312.262,E2 -31312.262} C_VEL
LIN {X 0,Y 52.961,Z 602.338,A -85,B 0,C 180,E1 -31314.422,E2 -31314.422} C_VEL
LIN {X 0,Y 65.164,Z 595.217,A -85,B 0,C 180,E1 -31316.053,E2 -31316.053} C_VEL
LIN {X 0,Y 70.413,Z 591.649,A -85,B 0,C 180,E1 -31316.487,E2 -31316.487} C_VEL
LIN {X 0,Y 70.388,Z 591.674,A -85,B 0,C 180,E1 -31316.829,E2 -31316.829} C_VEL
LIN {X 0,Y 58.015,Z 599.623,A -85,B 0,C 180,E1 -31318.052,E2 -31318.052} C_VEL
LIN {X 0,Y 44.65,Z 606.487,A -85,B 0,C 180,E1 -31319.997,E2 -31319.997} C_VEL
LIN {X 0,Y 31.69,Z 611.666,A -85,B 0,C 180,E1 -31323.63,E2 -31323.63} C_VEL
LIN {X 0,Y 21.353,Z 614.836,A -85,B 0,C 180,E1 -31329.111,E2 -31329.111} C_VEL
LIN {X 0,Y 8.696,Z 617.804,A -85,B 0,C 180,E1 -31356.085,E2 -31356.085} C_VEL
LIN {X 0,Y 5.727,Z 618.762,A -85,B 0,C 180,E1 -31410.003,E2 -31410.003} C_VEL
LIN {X 0,Y 8.745,Z 619.348,A -85,B 0,C 180,E1 -31463.481,E2 -31463.481} C_VEL
LIN {X 0,Y 21.379,Z 619.519,A -85,B 0,C 180,E1 -31490.479,E2 -31490.479} C_VEL
LIN {X 0,Y 35.186,Z 618.383,A -85,B 0,C 180,E1 -31497.075,E2 -31497.075} C_VEL
LIN {X 0,Y 37.47,Z 618.056,A -85,B 0,C 180,E1 -31500.003,E2 -31500.003} C_VEL
LIN {X 0,Y 27.084,Z 619.058,A -85,B 0,C 180,E1 -31503.822,E2 -31503.822} C_VEL
LIN {X 0,Y 27.084,Z 619.058,A -85,B 0,C 180,E1 -31503.822,E2 -31503.822}

QRS_NEXT_CUT()

QRS_NEXT()
QRS_HOME()

END
